KUKA KRL program: EPS_2_25694_GD04_A_20260114065903.src

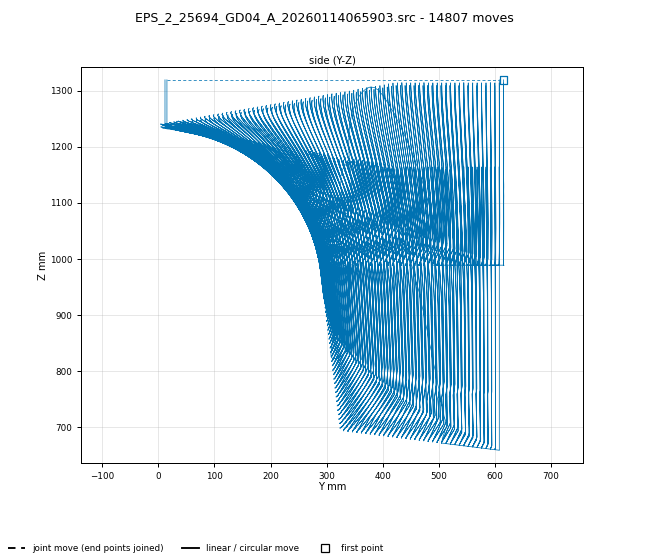
[picture p0: tool path of EPS_2_25694_GD04_A_20260114065903.src, 14807 of 14809 moves have a stored position in this frame; points joined in program order, loops and branches not executed]
&ACCESS RVP
&REL 4
&COMMENT QRS 19112012
&PARAM EDITMASK = *
DEF PART()
EXT BAS (BAS_COMMAND :IN,REAL :IN )
INT I
BAS (#INITMOV,0 )

;KUKA QRS Post kuka4.cps  Date:22-06-2017 !

File_ID=2971

QRS_PRE_INIT()

;Init var - Until changes are made in qrs_pre_init
Outlet_Square_prg=0
Inlet_1_Square_prg=0
Inlet_2_Square_prg=0
Inlet_3_Square_prg=0
Inlet_4_Square_prg=0
Inlet_5_Square_prg=0

Outlet_1={X 0.000, Y 425.000, Z 1043.000, B 0.000, E1 0.000 }
Inlet_1={X 0.000, Y 425.000, Z 703.000, B 0.000, E1 180.000 }
Outlet_1_type=533
Inlet_1_type=533
;QRS#1=Sidecore dimensions
;QRS#2=525-21" Concrete
;QRS#3=525-21" Concrete
;QRS#4=
;QRS#5=
;QRS#6=
;QRS#7=
;QRS#8=
;QRS#9=S306-32
;QRS#10=S306-32
;QRS#11=
;QRS#12=
;QRS#13=
;QRS#14=
;QRS#15=
;QRS#16=1220x127x1676 5,5'
;QRS#17=EPS Height
;QRS#18=1309,5
;QRS#19=*
;QRS#20= UPDATED VERSION 22-06-2017
;QRS#21=*
Outlet_Square=0250
Inlet_1_Square=0250
Inlet_2_Square=0
Inlet_3_Square=0
Inlet_4_Square=0
Inlet_5_Square=0
Mill_Square=1
Outlet_Square_Prg=263
Inlet_1_Square_prg=263

QRS_INIT()

$ADVANCE=5

; T1
PTP {E1 172.608,E2 172.608}
PTP {X 0,Y 615.419,A -85,B 0,C 180,E1 172.608,E2 172.608,E3 0,E4 0,E5 0,E6 0}
QRS_SPEED_INIT()
LIN {X 0,Y 615.419,Z 1319.5,A -85,B 0,C 180,E1 172.608,E2 172.608,E3 0,E4 0,E5 0,E6 0} C_VEL
LIN {X 0,Y 615.419,Z 991.03,A -85,B 0,C 180,E1 172.608,E2 172.608} C_VEL
LIN {X 0,Y 615.445,Z 989.03,A -85,B 0,C 180,E1 172.794,E2 172.794} C_VEL
LIN {X 0,Y 615.855,Z 989.03,A -85,B 0,C 180,E1 174.193,E2 174.193} C_VEL
LIN {X 0,Y 615.875,Z 989.03,A -85,B 0,C 180,E1 178.841,E2 178.841} C_VEL
LIN {X 0,Y 615.861,Z 989.03,A -85,B 0,C 180,E1 183.48,E2 183.48} C_VEL
LIN {X 0,Y 615.852,Z 989.03,A -85,B 0,C 180,E1 188.143,E2 188.143} C_VEL
LIN {X 0,Y 615.813,Z 989.03,A -85,B 0,C 180,E1 192.861,E2 192.861} C_VEL
LIN {X 0,Y 615.807,Z 989.03,A -85,B 0,C 180,E1 197.67,E2 197.67} C_VEL
LIN {X 0,Y 615.805,Z 989.03,A -85,B 0,C 180,E1 198.001,E2 198.001} C_VEL
LIN {X 0,Y 615.77,Z 989.03,A -85,B 0,C 180,E1 202.613,E2 202.613} C_VEL
LIN {X 0,Y 615.246,Z 989.03,A -85,B 0,C 180,E1 205.172,E2 205.172} C_VEL
LIN {X 0,Y 615.74,Z 989.03,A -85,B 0,C 180,E1 207.741,E2 207.741} C_VEL
LIN {X 0,Y 615.245,Z 989.03,A -85,B 0,C 180,E1 210.422,E2 210.422} C_VEL
LIN {X 0,Y 615.834,Z 989.03,A -85,B 0,C 180,E1 213.117,E2 213.117} C_VEL
LIN {X 0,Y 615.539,Z 989.03,A -85,B 0,C 180,E1 215.951,E2 215.951} C_VEL
LIN {X 0,Y 615.602,Z 989.03,A -85,B 0,C 180,E1 217.868,E2 217.868} C_VEL
LIN {X 0,Y 615.676,Z 989.03,A -85,B 0,C 180,E1 221.907,E2 221.907} C_VEL
LIN {X 0,Y 615.231,Z 989.03,A -85,B 0,C 180,E1 225.147,E2 225.147} C_VEL
LIN {X 0,Y 615.682,Z 989.03,A -85,B 0,C 180,E1 228.095,E2 228.095} C_VEL
LIN {X 0,Y 615.612,Z 989.03,A -85,B 0,C 180,E1 232.134,E2 232.134} C_VEL
LIN {X 0,Y 615.586,Z 989.03,A -85,B 0,C 180,E1 234.054,E2 234.054} C_VEL
LIN {X 0,Y 615.729,Z 989.03,A -85,B 0,C 180,E1 236.076,E2 236.076} C_VEL
LIN {X 0,Y 615.766,Z 989.03,A -85,B 0,C 180,E1 236.881,E2 236.881} C_VEL
LIN {X 0,Y 615.665,Z 989.03,A -85,B 0,C 180,E1 239.603,E2 239.603} C_VEL
LIN {X 0,Y 615.571,Z 989.03,A -85,B 0,C 180,E1 240.51,E2 240.51} C_VEL
LIN {X 0,Y 615.286,Z 989.03,A -85,B 0,C 180,E1 240.561,E2 240.561} C_VEL
LIN {X 0,Y 615.222,Z 991.746,A -85,B 0,C 180,E1 240.607,E2 240.607} C_VEL
LIN {X 0,Y 615.448,Z 1058.521,A -85,B 0,C 180,E1 241.501,E2 241.501} C_VEL
LIN {X 0,Y 615.53,Z 1069.288,A -85,B 0,C 180,E1 241.68,E2 241.68} C_VEL
LIN {X 0,Y 615.536,Z 1083.605,A -85,B 0,C 180,E1 241.986,E2 241.986} C_VEL
LIN {X 0,Y 615.507,Z 1092.707,A -85,B 0,C 180,E1 242.216,E2 242.216} C_VEL
LIN {X 0,Y 615.685,Z 1108.532,A -85,B 0,C 180,E1 242.707,E2 242.707} C_VEL
LIN {X 0,Y 615.645,Z 1120.963,A -85,B 0,C 180,E1 243.153,E2 243.153} C_VEL
LIN {X 0,Y 615.565,Z 1130.88,A -85,B 0,C 180,E1 243.554,E2 243.554} C_VEL
LIN {X 0,Y 615.702,Z 1146.604,A -85,B 0,C 180,E1 244.287,E2 244.287} C_VEL
LIN {X 0,Y 615.674,Z 1158.954,A -85,B 0,C 180,E1 244.936,E2 244.936} C_VEL
LIN {X 0,Y 615.686,Z 1170.579,A -85,B 0,C 180,E1 245.615,E2 245.615} C_VEL
LIN {X 0,Y 615.71,Z 1182.431,A -85,B 0,C 180,E1 246.381,E2 246.381} C_VEL
LIN {X 0,Y 615.719,Z 1193.096,A -85,B 0,C 180,E1 247.136,E2 247.136} C_VEL
LIN {X 0,Y 615.717,Z 1204.396,A -85,B 0,C 180,E1 248.013,E2 248.013} C_VEL
LIN {X 0,Y 615.705,Z 1213.657,A -85,B 0,C 180,E1 248.792,E2 248.792} C_VEL
LIN {X 0,Y 615.754,Z 1223.794,A -85,B 0,C 180,E1 249.723,E2 249.723} C_VEL
LIN {X 0,Y 615.723,Z 1233.057,A -85,B 0,C 180,E1 250.647,E2 250.647} C_VEL
LIN {X 0,Y 615.68,Z 1241.424,A -85,B 0,C 180,E1 251.549,E2 251.549} C_VEL
LIN {X 0,Y 615.758,Z 1249.778,A -85,B 0,C 180,E1 252.532,E2 252.532} C_VEL
LIN {X 0,Y 615.711,Z 1257.683,A -85,B 0,C 180,E1 253.542,E2 253.542} C_VEL
LIN {X 0,Y 615.578,Z 1264.428,A -85,B 0,C 180,E1 254.473,E2 254.473} C_VEL
LIN {X 0,Y 615.673,Z 1272.062,A -85,B 0,C 180,E1 255.645,E2 255.645} C_VEL
LIN {X 0,Y 615.813,Z 1277.438,A -85,B 0,C 180,E1 256.544,E2 256.544} C_VEL
LIN {X 0,Y 615.579,Z 1283.91,A -85,B 0,C 180,E1 257.728,E2 257.728} C_VEL
LIN {X 0,Y 615.618,Z 1289.624,A -85,B 0,C 180,E1 258.913,E2 258.913} C_VEL
LIN {X 0,Y 615.829,Z 1294.634,A -85,B 0,C 180,E1 260.096,E2 260.096} C_VEL
LIN {X 0,Y 615.605,Z 1299.063,A -85,B 0,C 180,E1 261.268,E2 261.268} C_VEL
LIN {X 0,Y 615.656,Z 1303.46,A -85,B 0,C 180,E1 262.657,E2 262.657} C_VEL
LIN {X 0,Y 615.79,Z 1306.367,A -85,B 0,C 180,E1 263.748,E2 263.748} C_VEL
LIN {X 0,Y 615.529,Z 1309.384,A -85,B 0,C 180,E1 265.123,E2 265.123} C_VEL
LIN {X 0,Y 615.632,Z 1311.593,A -85,B 0,C 180,E1 266.519,E2 266.519} C_VEL
LIN {X 0,Y 615.819,Z 1312.67,A -85,B 0,C 180,E1 267.449,E2 267.449} C_VEL
LIN {X 0,Y 615.544,Z 1313.716,A -85,B 0,C 180,E1 268.84,E2 268.84} C_VEL
LIN {X 0,Y 615.841,Z 1313.659,A -85,B 0,C 180,E1 271.159,E2 271.159} C_VEL
LIN {X 0,Y 615.625,Z 1313.07,A -85,B 0,C 180,E1 272.088,E2 272.088} C_VEL
LIN {X 0,Y 615.537,Z 1311.611,A -85,B 0,C 180,E1 273.482,E2 273.482} C_VEL
LIN {X 0,Y 615.808,Z 1309.333,A -85,B 0,C 180,E1 274.875,E2 274.875} C_VEL
LIN {X 0,Y 615.603,Z 1306.409,A -85,B 0,C 180,E1 276.25,E2 276.25} C_VEL
LIN {X 0,Y 615.617,Z 1303.276,A -85,B 0,C 180,E1 277.415,E2 277.415} C_VEL
LIN {X 0,Y 615.787,Z 1299.035,A -85,B 0,C 180,E1 278.729,E2 278.729} C_VEL
LIN {X 0,Y 615.576,Z 1294.671,A -85,B 0,C 180,E1 279.908,E2 279.908} C_VEL
LIN {X 0,Y 615.636,Z 1289.622,A -85,B 0,C 180,E1 281.086,E2 281.086} C_VEL
LIN {X 0,Y 615.811,Z 1283.883,A -85,B 0,C 180,E1 282.267,E2 282.267} C_VEL
LIN {X 0,Y 615.629,Z 1277.456,A -85,B 0,C 180,E1 283.46,E2 283.46} C_VEL
LIN {X 0,Y 615.698,Z 1270.195,A -85,B 0,C 180,E1 284.654,E2 284.654} C_VEL
LIN {X 0,Y 615.81,Z 1264.632,A -85,B 0,C 180,E1 285.488,E2 285.488} C_VEL
LIN {X 0,Y 615.663,Z 1255.2,A -85,B 0,C 180,E1 286.791,E2 286.791} C_VEL
LIN {X 0,Y 615.737,Z 1246.606,A -85,B 0,C 180,E1 287.852,E2 287.852} C_VEL
LIN {X 0,Y 615.77,Z 1238.414,A -85,B 0,C 180,E1 288.784,E2 288.784} C_VEL
LIN {X 0,Y 615.695,Z 1228.526,A -85,B 0,C 180,E1 289.816,E2 289.816} C_VEL
LIN {X 0,Y 615.712,Z 1220.54,A -85,B 0,C 180,E1 290.588,E2 290.588} C_VEL
LIN {X 0,Y 615.743,Z 1210.038,A -85,B 0,C 180,E1 291.518,E2 291.518} C_VEL
LIN {X 0,Y 615.702,Z 1200.053,A -85,B 0,C 180,E1 292.335,E2 292.335} C_VEL
LIN {X 0,Y 615.701,Z 1190.291,A -85,B 0,C 180,E1 293.071,E2 293.071} C_VEL
LIN {X 0,Y 615.684,Z 1178.615,A -85,B 0,C 180,E1 293.875,E2 293.875} C_VEL
LIN {X 0,Y 615.706,Z 1166.573,A -85,B 0,C 180,E1 294.624,E2 294.624} C_VEL
LIN {X 0,Y 615.664,Z 1155.895,A -85,B 0,C 180,E1 295.233,E2 295.233} C_VEL
LIN {X 0,Y 615.663,Z 1145.03,A -85,B 0,C 180,E1 295.795,E2 295.795} C_VEL
LIN {X 0,Y 615.698,Z 1130.88,A -85,B 0,C 180,E1 296.439,E2 296.439} C_VEL
LIN {X 0,Y 615.617,Z 1117.679,A -85,B 0,C 180,E1 296.971,E2 296.971} C_VEL
LIN {X 0,Y 615.552,Z 1108.531,A -85,B 0,C 180,E1 297.299,E2 297.299} C_VEL
LIN {X 0,Y 615.614,Z 1091.815,A -85,B 0,C 180,E1 297.801,E2 297.801} C_VEL
LIN {X 0,Y 615.471,Z 1080.012,A -85,B 0,C 180,E1 298.104,E2 298.104} C_VEL
LIN {X 0,Y 615.643,Z 1066.85,A -85,B 0,C 180,E1 298.361,E2 298.361} C_VEL
LIN {X 0,Y 615.612,Z 1048.004,A -85,B 0,C 180,E1 298.638,E2 298.638} C_VEL
LIN {X 0,Y 615.269,Z 989.03,A -85,B 0,C 180,E1 299.434,E2 299.434} C_VEL
LIN {X 0,Y 615.512,Z 989.03,A -85,B 0,C 180,E1 299.476,E2 299.476} C_VEL
LIN {X 0,Y 615.842,Z 989.03,A -85,B 0,C 180,E1 300.388,E2 300.388} C_VEL
LIN {X 0,Y 615.705,Z 989.03,A -85,B 0,C 180,E1 305.938,E2 305.938} C_VEL
LIN {X 0,Y 615.769,Z 989.03,A -85,B 0,C 180,E1 308.853,E2 308.853} C_VEL
LIN {X 0,Y 615.266,Z 989.03,A -85,B 0,C 180,E1 311.939,E2 311.939} C_VEL
LIN {X 0,Y 615.689,Z 989.03,A -85,B 0,C 180,E1 314.896,E2 314.896} C_VEL
LIN {X 0,Y 615.648,Z 989.03,A -85,B 0,C 180,E1 318.494,E2 318.494} C_VEL
LIN {X 0,Y 615.37,Z 989.03,A -85,B 0,C 180,E1 321.115,E2 321.115} C_VEL
LIN {X 0,Y 615.425,Z 989.03,A -85,B 0,C 180,E1 322.154,E2 322.154} C_VEL
LIN {X 0,Y 615.683,Z 989.03,A -85,B 0,C 180,E1 324.059,E2 324.059} C_VEL
LIN {X 0,Y 615.149,Z 989.03,A -85,B 0,C 180,E1 326.842,E2 326.842} C_VEL
LIN {X 0,Y 615.748,Z 989.03,A -85,B 0,C 180,E1 329.606,E2 329.606} C_VEL
LIN {X 0,Y 615.235,Z 989.03,A -85,B 0,C 180,E1 332.234,E2 332.234} C_VEL
LIN {X 0,Y 615.77,Z 989.03,A -85,B 0,C 180,E1 334.851,E2 334.851} C_VEL
LIN {X 0,Y 615.796,Z 989.03,A -85,B 0,C 180,E1 339.878,E2 339.878} C_VEL
LIN {X 0,Y 615.802,Z 989.03,A -85,B 0,C 180,E1 343.784,E2 343.784} C_VEL
LIN {X 0,Y 615.822,Z 989.03,A -85,B 0,C 180,E1 349.507,E2 349.507} C_VEL
LIN {X 0,Y 615.853,Z 989.03,A -85,B 0,C 180,E1 354.193,E2 354.193} C_VEL
LIN {X 0,Y 615.865,Z 989.03,A -85,B 0,C 180,E1 358.841,E2 358.841} C_VEL
LIN {X 0,Y 615.866,Z 989.03,A -85,B 0,C 180,E1 363.48,E2 363.48} C_VEL
LIN {X 0,Y 615.845,Z 989.03,A -85,B 0,C 180,E1 368.143,E2 368.143} C_VEL
LIN {X 0,Y 615.803,Z 989.03,A -85,B 0,C 180,E1 372.862,E2 372.862} C_VEL
LIN {X 0,Y 615.806,Z 989.03,A -85,B 0,C 180,E1 377.67,E2 377.67} C_VEL
LIN {X 0,Y 615.804,Z 989.03,A -85,B 0,C 180,E1 378.001,E2 378.001} C_VEL
LIN {X 0,Y 615.787,Z 989.03,A -85,B 0,C 180,E1 382.612,E2 382.612} C_VEL
LIN {X 0,Y 615.244,Z 989.03,A -85,B 0,C 180,E1 385.172,E2 385.172} C_VEL
LIN {X 0,Y 615.735,Z 989.03,A -85,B 0,C 180,E1 387.741,E2 387.741} C_VEL
LIN {X 0,Y 615.177,Z 989.03,A -85,B 0,C 180,E1 390.425,E2 390.425} C_VEL
LIN {X 0,Y 615.705,Z 989.03,A -85,B 0,C 180,E1 393.124,E2 393.124} C_VEL
LIN {X 0,Y 615.645,Z 989.03,A -85,B 0,C 180,E1 393.916,E2 393.916} C_VEL
LIN {X 0,Y 615.651,Z 989.03,A -85,B 0,C 180,E1 398.864,E2 398.864} C_VEL
LIN {X 0,Y 615.251,Z 989.03,A -85,B 0,C 180,E1 401.943,E2 401.943} C_VEL
LIN {X 0,Y 615.678,Z 989.03,A -85,B 0,C 180,E1 404.897,E2 404.897} C_VEL
LIN {X 0,Y 615.658,Z 989.03,A -85,B 0,C 180,E1 408.496,E2 408.496} C_VEL
LIN {X 0,Y 615.375,Z 989.03,A -85,B 0,C 180,E1 411.117,E2 411.117} C_VEL
LIN {X 0,Y 615.426,Z 989.03,A -85,B 0,C 180,E1 412.156,E2 412.156} C_VEL
LIN {X 0,Y 615.691,Z 989.03,A -85,B 0,C 180,E1 414.061,E2 414.061} C_VEL
LIN {X 0,Y 615.154,Z 989.03,A -85,B 0,C 180,E1 416.844,E2 416.844} C_VEL
LIN {X 0,Y 615.773,Z 989.03,A -85,B 0,C 180,E1 419.609,E2 419.609} C_VEL
LIN {X 0,Y 615.759,Z 989.03,A -85,B 0,C 180,E1 423.303,E2 423.303} C_VEL
LIN {X 0,Y 615.27,Z 989.079,A -85,B 0,C 180,E1 423.866,E2 423.866} C_VEL
LIN {X 0,Y 615.494,Z 997.667,A -85,B 0,C 180,E1 424.288,E2 424.288} C_VEL
LIN {X 0,Y 615.612,Z 1009.734,A -85,B 0,C 180,E1 424.933,E2 424.933} C_VEL
LIN {X 0,Y 615.672,Z 1021.343,A -85,B 0,C 180,E1 425.618,E2 425.618} C_VEL
LIN {X 0,Y 615.7,Z 1032.734,A -85,B 0,C 180,E1 426.357,E2 426.357} C_VEL
LIN {X 0,Y 615.717,Z 1042.488,A -85,B 0,C 180,E1 427.044,E2 427.044} C_VEL
LIN {X 0,Y 615.706,Z 1053.812,A -85,B 0,C 180,E1 427.919,E2 427.919} C_VEL
LIN {X 0,Y 615.708,Z 1064.155,A -85,B 0,C 180,E1 428.792,E2 428.792} C_VEL
LIN {X 0,Y 615.732,Z 1072.675,A -85,B 0,C 180,E1 429.568,E2 429.568} C_VEL
LIN {X 0,Y 615.739,Z 1082.034,A -85,B 0,C 180,E1 430.493,E2 430.493} C_VEL
LIN {X 0,Y 615.681,Z 1089.889,A -85,B 0,C 180,E1 431.327,E2 431.327} C_VEL
LIN {X 0,Y 615.735,Z 1098.523,A -85,B 0,C 180,E1 432.328,E2 432.328} C_VEL
LIN {X 0,Y 615.758,Z 1106.541,A -85,B 0,C 180,E1 433.341,E2 433.341} C_VEL
LIN {X 0,Y 615.587,Z 1114.528,A -85,B 0,C 180,E1 434.443,E2 434.443} C_VEL
LIN {X 0,Y 615.629,Z 1120.5,A -85,B 0,C 180,E1 435.344,E2 435.344} C_VEL
LIN {X 0,Y 615.814,Z 1127.695,A -85,B 0,C 180,E1 436.544,E2 436.544} C_VEL
LIN {X 0,Y 615.591,Z 1134.13,A -85,B 0,C 180,E1 437.729,E2 437.729} C_VEL
LIN {X 0,Y 615.618,Z 1139.819,A -85,B 0,C 180,E1 438.913,E2 438.913} C_VEL
LIN {X 0,Y 615.817,Z 1144.809,A -85,B 0,C 180,E1 440.096,E2 440.096} C_VEL
LIN {X 0,Y 615.604,Z 1149.222,A -85,B 0,C 180,E1 441.268,E2 441.268} C_VEL
LIN {X 0,Y 615.654,Z 1153.586,A -85,B 0,C 180,E1 442.659,E2 442.659} C_VEL
LIN {X 0,Y 615.797,Z 1156.474,A -85,B 0,C 180,E1 443.747,E2 443.747} C_VEL
LIN {X 0,Y 615.543,Z 1159.456,A -85,B 0,C 180,E1 445.123,E2 445.123} C_VEL
LIN {X 0,Y 615.553,Z 1161.021,A -85,B 0,C 180,E1 446.053,E2 446.053} C_VEL
LIN {X 0,Y 615.633,Z 1161.646,A -85,B 0,C 180,E1 446.519,E2 446.519} C_VEL
LIN {X 0,Y 615.703,Z 1163.087,A -85,B 0,C 180,E1 447.912,E2 447.912} C_VEL
LIN {X 0,Y 615.545,Z 1163.726,A -85,B 0,C 180,E1 448.84,E2 448.84} C_VEL
LIN {X 0,Y 615.84,Z 1163.646,A -85,B 0,C 180,E1 451.159,E2 451.159} C_VEL
LIN {X 0,Y 615.601,Z 1162.656,A -85,B 0,C 180,E1 452.552,E2 452.552} C_VEL
LIN {X 0,Y 615.611,Z 1161.544,A -85,B 0,C 180,E1 453.481,E2 453.481} C_VEL
LIN {X 0,Y 615.797,Z 1159.26,A -85,B 0,C 180,E1 454.875,E2 454.875} C_VEL
LIN {X 0,Y 615.534,Z 1156.318,A -85,B 0,C 180,E1 456.245,E2 456.245} C_VEL
LIN {X 0,Y 615.586,Z 1153.213,A -85,B 0,C 180,E1 457.395,E2 457.395} C_VEL
LIN {X 0,Y 615.789,Z 1148.868,A -85,B 0,C 180,E1 458.729,E2 458.729} C_VEL
LIN {X 0,Y 615.587,Z 1144.486,A -85,B 0,C 180,E1 459.908,E2 459.908} C_VEL
LIN {X 0,Y 615.631,Z 1139.418,A -85,B 0,C 180,E1 461.086,E2 461.086} C_VEL
LIN {X 0,Y 615.804,Z 1133.652,A -85,B 0,C 180,E1 462.267,E2 462.267} C_VEL
LIN {X 0,Y 615.622,Z 1127.187,A -85,B 0,C 180,E1 463.46,E2 463.46} C_VEL
LIN {X 0,Y 615.693,Z 1119.896,A -85,B 0,C 180,E1 464.654,E2 464.654} C_VEL
LIN {X 0,Y 615.77,Z 1112.739,A -85,B 0,C 180,E1 465.717,E2 465.717} C_VEL
LIN {X 0,Y 615.611,Z 1104.213,A -85,B 0,C 180,E1 466.871,E2 466.871} C_VEL
LIN {X 0,Y 615.662,Z 1096.204,A -85,B 0,C 180,E1 467.856,E2 467.856} C_VEL
LIN {X 0,Y 615.759,Z 1088.025,A -85,B 0,C 180,E1 468.781,E2 468.781} C_VEL
LIN {X 0,Y 615.689,Z 1079.643,A -85,B 0,C 180,E1 469.662,E2 469.662} C_VEL
LIN {X 0,Y 615.685,Z 1070.04,A -85,B 0,C 180,E1 470.589,E2 470.589} C_VEL
LIN {X 0,Y 615.724,Z 1059.495,A -85,B 0,C 180,E1 471.519,E2 471.519} C_VEL
LIN {X 0,Y 615.715,Z 1049.452,A -85,B 0,C 180,E1 472.335,E2 472.335} C_VEL
LIN {X 0,Y 615.709,Z 1039.629,A -85,B 0,C 180,E1 473.072,E2 473.072} C_VEL
LIN {X 0,Y 615.662,Z 1027.858,A -85,B 0,C 180,E1 473.878,E2 473.878} C_VEL
LIN {X 0,Y 615.718,Z 1017.248,A -85,B 0,C 180,E1 474.54,E2 474.54} C_VEL
LIN {X 0,Y 615.706,Z 1005.438,A -85,B 0,C 180,E1 475.21,E2 475.21} C_VEL
LIN {X 0,Y 615.597,Z 993.583,A -85,B 0,C 180,E1 475.821,E2 475.821} C_VEL
LIN {X 0,Y 615.42,Z 990.651,A -85,B 0,C 180,E1 475.964,E2 475.964} C_VEL
LIN {X 0,Y 615.152,Z 989.03,A -85,B 0,C 180,E1 476.061,E2 476.061} C_VEL
LIN {X 0,Y 615.489,Z 989.03,A -85,B 0,C 180,E1 476.139,E2 476.139} C_VEL
LIN {X 0,Y 615.881,Z 989.03,A -85,B 0,C 180,E1 476.434,E2 476.434} C_VEL
LIN {X 0,Y 615.828,Z 989.03,A -85,B 0,C 180,E1 477.736,E2 477.736} C_VEL
LIN {X 0,Y 615.182,Z 989.03,A -85,B 0,C 180,E1 480.424,E2 480.424} C_VEL
LIN {X 0,Y 615.708,Z 989.03,A -85,B 0,C 180,E1 483.123,E2 483.123} C_VEL
LIN {X 0,Y 615.642,Z 989.03,A -85,B 0,C 180,E1 483.912,E2 483.912} C_VEL
LIN {X 0,Y 615.656,Z 989.03,A -85,B 0,C 180,E1 488.862,E2 488.862} C_VEL
LIN {X 0,Y 615.249,Z 989.03,A -85,B 0,C 180,E1 491.941,E2 491.941} C_VEL
LIN {X 0,Y 615.661,Z 989.03,A -85,B 0,C 180,E1 494.893,E2 494.893} C_VEL
LIN {X 0,Y 615.652,Z 989.03,A -85,B 0,C 180,E1 498.494,E2 498.494} C_VEL
LIN {X 0,Y 615.375,Z 989.03,A -85,B 0,C 180,E1 501.116,E2 501.116} C_VEL
LIN {X 0,Y 615.419,Z 989.03,A -85,B 0,C 180,E1 502.154,E2 502.154} C_VEL
LIN {X 0,Y 615.689,Z 989.03,A -85,B 0,C 180,E1 504.059,E2 504.059} C_VEL
LIN {X 0,Y 615.154,Z 989.03,A -85,B 0,C 180,E1 506.842,E2 506.842} C_VEL
LIN {X 0,Y 615.751,Z 989.03,A -85,B 0,C 180,E1 509.606,E2 509.606} C_VEL
LIN {X 0,Y 615.246,Z 989.03,A -85,B 0,C 180,E1 512.235,E2 512.235} C_VEL
LIN {X 0,Y 615.777,Z 989.03,A -85,B 0,C 180,E1 514.851,E2 514.851} C_VEL
LIN {X 0,Y 615.807,Z 989.03,A -85,B 0,C 180,E1 519.879,E2 519.879} C_VEL
LIN {X 0,Y 615.758,Z 989.03,A -85,B 0,C 180,E1 523.299,E2 523.299} C_VEL
LIN {X 0,Y 615.415,Z 989.03,A -85,B 0,C 180,E1 524.738,E2 524.738} C_VEL
LIN {X 0,Y 615.826,Z 989.03,A -85,B 0,C 180,E1 529.507,E2 529.507} C_VEL
LIN {X 0,Y 615.445,Z 989.03,A -85,B 0,C 180,E1 532.794,E2 532.794} C_VEL
LIN {X 0,Y 613.023,Z 989.03,A -85,B 0,C 180,E1 533.996,E2 533.996} C_VEL
LIN {X 0,Y 607.607,Z 989.03,A -85,B 0,C 180,E1 535.793,E2 535.793} C_VEL
LIN {X 0,Y 607.497,Z 989.03,A -85,B 0,C 180,E1 536.001,E2 536.001} C_VEL
LIN {X 0,Y 607.621,Z 989.03,A -85,B 0,C 180,E1 540,E2 540} C_VEL
LIN {X 0,Y 607.699,Z 989.03,A -85,B 0,C 180,E1 544.272,E2 544.272} C_VEL
LIN {X 0,Y 607.796,Z 989.03,A -85,B 0,C 180,E1 548.567,E2 548.567} C_VEL
LIN {X 0,Y 607.904,Z 989.03,A -85,B 0,C 180,E1 552.909,E2 552.909} C_VEL
LIN {X 0,Y 607.63,Z 989.03,A -85,B 0,C 180,E1 558.834,E2 558.834} C_VEL
LIN {X 0,Y 607.589,Z 989.03,A -85,B 0,C 180,E1 563.413,E2 563.413} C_VEL
LIN {X 0,Y 607.696,Z 989.03,A -85,B 0,C 180,E1 568.15,E2 568.15} C_VEL
LIN {X 0,Y 607.93,Z 989.03,A -85,B 0,C 180,E1 573.097,E2 573.097} C_VEL
LIN {X 0,Y 607.556,Z 989.03,A -85,B 0,C 180,E1 578.382,E2 578.382} C_VEL
LIN {X 0,Y 607.691,Z 989.03,A -85,B 0,C 180,E1 582.1,E2 582.1} C_VEL
LIN {X 0,Y 607.775,Z 989.03,A -85,B 0,C 180,E1 588.144,E2 588.144} C_VEL
LIN {X 0,Y 607.625,Z 989.03,A -85,B 0,C 180,E1 593.413,E2 593.413} C_VEL
LIN {X 0,Y 607.652,Z 989.03,A -85,B 0,C 180,E1 598.566,E2 598.566} C_VEL
LIN {X 0,Y 607.709,Z 989.03,A -85,B 0,C 180,E1 600.165,E2 600.165} C_VEL
LIN {X 0,Y 608.575,Z 1077.126,A -85,B 0,C 180,E1 601.489,E2 601.489} C_VEL
LIN {X 0,Y 608.555,Z 1114.756,A -85,B 0,C 180,E1 602.585,E2 602.585} C_VEL
LIN {X 0,Y 608.428,Z 1150.792,A -85,B 0,C 180,E1 604.177,E2 604.177} C_VEL
LIN {X 0,Y 608.274,Z 1185.935,A -85,B 0,C 180,E1 606.322,E2 606.322} C_VEL
LIN {X 0,Y 608.111,Z 1217.995,A -85,B 0,C 180,E1 608.911,E2 608.911} C_VEL
LIN {X 0,Y 607.969,Z 1246.718,A -85,B 0,C 180,E1 611.925,E2 611.925} C_VEL
LIN {X 0,Y 607.835,Z 1271.188,A -85,B 0,C 180,E1 615.295,E2 615.295} C_VEL
LIN {X 0,Y 607.763,Z 1290.437,A -85,B 0,C 180,E1 618.905,E2 618.905} C_VEL
LIN {X 0,Y 607.783,Z 1303.716,A -85,B 0,C 180,E1 622.51,E2 622.51} C_VEL
LIN {X 0,Y 607.66,Z 1310.955,A -85,B 0,C 180,E1 625.727,E2 625.727} C_VEL
LIN {X 0,Y 607.699,Z 1314.085,A -85,B 0,C 180,E1 628.577,E2 628.577} C_VEL
LIN {X 0,Y 607.887,Z 1314.086,A -85,B 0,C 180,E1 631.422,E2 631.422} C_VEL
LIN {X 0,Y 607.907,Z 1309.758,A -85,B 0,C 180,E1 634.984,E2 634.984} C_VEL
LIN {X 0,Y 607.881,Z 1299.074,A -85,B 0,C 180,E1 638.925,E2 638.925} C_VEL
LIN {X 0,Y 607.91,Z 1283.453,A -85,B 0,C 180,E1 642.544,E2 642.544} C_VEL
LIN {X 0,Y 607.956,Z 1262.352,A -85,B 0,C 180,E1 646.029,E2 646.029} C_VEL
LIN {X 0,Y 608.033,Z 1236.204,A -85,B 0,C 180,E1 649.27,E2 649.27} C_VEL
LIN {X 0,Y 608.169,Z 1206.028,A -85,B 0,C 180,E1 652.137,E2 652.137} C_VEL
LIN {X 0,Y 608.322,Z 1172.896,A -85,B 0,C 180,E1 654.55,E2 654.55} C_VEL
LIN {X 0,Y 608.503,Z 1136.751,A -85,B 0,C 180,E1 656.511,E2 656.511} C_VEL
LIN {X 0,Y 608.582,Z 1099.984,A -85,B 0,C 180,E1 657.91,E2 657.91} C_VEL
LIN {X 0,Y 608.716,Z 1064.141,A -85,B 0,C 180,E1 658.756,E2 658.756} C_VEL
LIN {X 0,Y 607.728,Z 989.475,A -85,B 0,C 180,E1 659.822,E2 659.822} C_VEL
LIN {X 0,Y 607.714,Z 989.03,A -85,B 0,C 180,E1 666.579,E2 666.579} C_VEL
LIN {X 0,Y 607.344,Z 989.03,A -85,B 0,C 180,E1 672.132,E2 672.132} C_VEL
LIN {X 0,Y 607.668,Z 989.03,A -85,B 0,C 180,E1 678.157,E2 678.157} C_VEL
LIN {X 0,Y 607.639,Z 989.03,A -85,B 0,C 180,E1 683.417,E2 683.417} C_VEL
LIN {X 0,Y 607.57,Z 989.03,A -85,B 0,C 180,E1 690.375,E2 690.375} C_VEL
LIN {X 0,Y 607.806,Z 989.03,A -85,B 0,C 180,E1 695.036,E2 695.036} C_VEL
LIN {X 0,Y 607.665,Z 989.03,A -85,B 0,C 180,E1 700.673,E2 700.673} C_VEL
LIN {X 0,Y 607.268,Z 989.03,A -85,B 0,C 180,E1 705.612,E2 705.612} C_VEL
LIN {X 0,Y 607.749,Z 989.03,A -85,B 0,C 180,E1 709.991,E2 709.991} C_VEL
LIN {X 0,Y 607.925,Z 989.03,A -85,B 0,C 180,E1 714.302,E2 714.302} C_VEL
LIN {X 0,Y 607.586,Z 989.03,A -85,B 0,C 180,E1 720,E2 720} C_VEL
LIN {X 0,Y 607.674,Z 989.03,A -85,B 0,C 180,E1 724.272,E2 724.272} C_VEL
LIN {X 0,Y 607.794,Z 989.03,A -85,B 0,C 180,E1 728.567,E2 728.567} C_VEL
LIN {X 0,Y 607.876,Z 989.03,A -85,B 0,C 180,E1 732.909,E2 732.909} C_VEL
LIN {X 0,Y 607.604,Z 989.03,A -85,B 0,C 180,E1 738.835,E2 738.835} C_VEL
LIN {X 0,Y 607.594,Z 989.03,A -85,B 0,C 180,E1 743.413,E2 743.413} C_VEL
LIN {X 0,Y 607.67,Z 989.03,A -85,B 0,C 180,E1 748.151,E2 748.151} C_VEL
LIN {X 0,Y 607.806,Z 989.03,A -85,B 0,C 180,E1 753.105,E2 753.105} C_VEL
LIN {X 0,Y 607.48,Z 989.03,A -85,B 0,C 180,E1 759.642,E2 759.642} C_VEL
LIN {X 0,Y 607.554,Z 989.03,A -85,B 0,C 180,E1 765.938,E2 765.938} C_VEL
LIN {X 0,Y 607.425,Z 989.03,A -85,B 0,C 180,E1 770.362,E2 770.362} C_VEL
LIN {X 0,Y 607.428,Z 989.03,A -85,B 0,C 180,E1 775.154,E2 775.154} C_VEL
LIN {X 0,Y 607.687,Z 989.03,A -85,B 0,C 180,E1 780.352,E2 780.352} C_VEL
LIN {X 0,Y 607.651,Z 989.82,A -85,B 0,C 180,E1 783.548,E2 783.548} C_VEL
LIN {X 0,Y 608.277,Z 1025.109,A -85,B 0,C 180,E1 785.545,E2 785.545} C_VEL
LIN {X 0,Y 608.154,Z 1058.841,A -85,B 0,C 180,E1 788.054,E2 788.054} C_VEL
LIN {X 0,Y 607.98,Z 1089.393,A -85,B 0,C 180,E1 791.027,E2 791.027} C_VEL
LIN {X 0,Y 607.797,Z 1115.33,A -85,B 0,C 180,E1 794.355,E2 794.355} C_VEL
LIN {X 0,Y 607.772,Z 1133.695,A -85,B 0,C 180,E1 797.453,E2 797.453} C_VEL
LIN {X 0,Y 607.781,Z 1149.241,A -85,B 0,C 180,E1 801.073,E2 801.073} C_VEL
LIN {X 0,Y 607.774,Z 1158.319,A -85,B 0,C 180,E1 804.301,E2 804.301} C_VEL
LIN {X 0,Y 607.769,Z 1162.96,A -85,B 0,C 180,E1 807.154,E2 807.154} C_VEL
LIN {X 0,Y 607.73,Z 1164.496,A -85,B 0,C 180,E1 810.001,E2 810.001} C_VEL
LIN {X 0,Y 607.709,Z 1162.852,A -85,B 0,C 180,E1 812.847,E2 812.847} C_VEL
LIN {X 0,Y 607.722,Z 1158.121,A -85,B 0,C 180,E1 815.701,E2 815.701} C_VEL
LIN {X 0,Y 607.813,Z 1147.564,A -85,B 0,C 180,E1 819.287,E2 819.287} C_VEL
LIN {X 0,Y 607.839,Z 1131.246,A -85,B 0,C 180,E1 822.911,E2 822.911} C_VEL
LIN {X 0,Y 607.898,Z 1110.686,A -85,B 0,C 180,E1 826.217,E2 826.217} C_VEL
LIN {X 0,Y 608.04,Z 1085.63,A -85,B 0,C 180,E1 829.286,E2 829.286} C_VEL
LIN {X 0,Y 608.175,Z 1055.481,A -85,B 0,C 180,E1 832.138,E2 832.138} C_VEL
LIN {X 0,Y 608.348,Z 1020.67,A -85,B 0,C 180,E1 834.648,E2 834.648} C_VEL
LIN {X 0,Y 607.948,Z 989.03,A -85,B 0,C 180,E1 836.439,E2 836.439} C_VEL
LIN {X 0,Y 607.81,Z 989.03,A -85,B 0,C 180,E1 843.107,E2 843.107} C_VEL
LIN {X 0,Y 607.506,Z 989.03,A -85,B 0,C 180,E1 849.647,E2 849.647} C_VEL
LIN {X 0,Y 607.518,Z 989.03,A -85,B 0,C 180,E1 855.936,E2 855.936} C_VEL
LIN {X 0,Y 607.424,Z 989.03,A -85,B 0,C 180,E1 860.366,E2 860.366} C_VEL
LIN {X 0,Y 607.422,Z 989.03,A -85,B 0,C 180,E1 865.155,E2 865.155} C_VEL
LIN {X 0,Y 607.567,Z 989.03,A -85,B 0,C 180,E1 870.378,E2 870.378} C_VEL
LIN {X 0,Y 607.799,Z 989.03,A -85,B 0,C 180,E1 875.036,E2 875.036} C_VEL
LIN {X 0,Y 607.663,Z 989.03,A -85,B 0,C 180,E1 881.167,E2 881.167} C_VEL
LIN {X 0,Y 607.249,Z 989.03,A -85,B 0,C 180,E1 885.733,E2 885.733} C_VEL
LIN {X 0,Y 607.754,Z 989.03,A -85,B 0,C 180,E1 889.991,E2 889.991} C_VEL
LIN {X 0,Y 607.909,Z 989.03,A -85,B 0,C 180,E1 894.302,E2 894.302} C_VEL
LIN {X 0,Y 607.497,Z 989.03,A -85,B 0,C 180,E1 896.001,E2 896.001} C_VEL
LIN {X 0,Y 603.696,Z 989.03,A -85,B 0,C 180,E1 897.613,E2 897.613} C_VEL
LIN {X 0,Y 599.806,Z 989.03,A -85,B 0,C 180,E1 899.244,E2 899.244} C_VEL
LIN {X 0,Y 599.78,Z 989.03,A -85,B 0,C 180,E1 904.329,E2 904.329} C_VEL
LIN {X 0,Y 599.852,Z 989.03,A -85,B 0,C 180,E1 908.681,E2 908.681} C_VEL
LIN {X 0,Y 599.925,Z 989.03,A -85,B 0,C 180,E1 913.083,E2 913.083} C_VEL
LIN {X 0,Y 599.672,Z 989.03,A -85,B 0,C 180,E1 919.094,E2 919.094} C_VEL
LIN {X 0,Y 599.598,Z 989.03,A -85,B 0,C 180,E1 923.744,E2 923.744} C_VEL
LIN {X 0,Y 599.687,Z 989.03,A -85,B 0,C 180,E1 928.56,E2 928.56} C_VEL
LIN {X 0,Y 599.814,Z 989.03,A -85,B 0,C 180,E1 933.878,E2 933.878} C_VEL
LIN {X 0,Y 599.539,Z 989.03,A -85,B 0,C 180,E1 938.992,E2 938.992} C_VEL
LIN {X 0,Y 599.496,Z 989.03,A -85,B 0,C 180,E1 943.115,E2 943.115} C_VEL
LIN {X 0,Y 599.595,Z 989.03,A -85,B 0,C 180,E1 949.129,E2 949.129} C_VEL
LIN {X 0,Y 599.717,Z 989.03,A -85,B 0,C 180,E1 954.638,E2 954.638} C_VEL
LIN {X 0,Y 599.889,Z 989.522,A -85,B 0,C 180,E1 959.748,E2 959.748} C_VEL
LIN {X 0,Y 601.492,Z 997.227,A -85,B 0,C 180,E1 959.942,E2 959.942} C_VEL
LIN {X 0,Y 601.63,Z 1077.166,A -85,B 0,C 180,E1 961.13,E2 961.13} C_VEL
LIN {X 0,Y 601.497,Z 1113.617,A -85,B 0,C 180,E1 962.194,E2 962.194} C_VEL
LIN {X 0,Y 601.209,Z 1148.932,A -85,B 0,C 180,E1 963.744,E2 963.744} C_VEL
LIN {X 0,Y 600.865,Z 1184.565,A -85,B 0,C 180,E1 965.914,E2 965.914} C_VEL
LIN {X 0,Y 600.542,Z 1217.043,A -85,B 0,C 180,E1 968.544,E2 968.544} C_VEL
LIN {X 0,Y 600.234,Z 1245.115,A -85,B 0,C 180,E1 971.494,E2 971.494} C_VEL
LIN {X 0,Y 599.993,Z 1269.748,A -85,B 0,C 180,E1 974.874,E2 974.874} C_VEL
LIN {X 0,Y 599.872,Z 1288.763,A -85,B 0,C 180,E1 978.39,E2 978.39} C_VEL
LIN {X 0,Y 599.857,Z 1301.445,A -85,B 0,C 180,E1 981.683,E2 981.683} C_VEL
LIN {X 0,Y 599.777,Z 1309.755,A -85,B 0,C 180,E1 984.948,E2 984.948} C_VEL
LIN {X 0,Y 599.8,Z 1314.085,A -85,B 0,C 180,E1 988.558,E2 988.558} C_VEL
LIN {X 0,Y 599.98,Z 1314.086,A -85,B 0,C 180,E1 991.441,E2 991.441} C_VEL
LIN {X 0,Y 599.994,Z 1309.758,A -85,B 0,C 180,E1 995.05,E2 995.05} C_VEL
LIN {X 0,Y 599.98,Z 1299.074,A -85,B 0,C 180,E1 999.044,E2 999.044} C_VEL
LIN {X 0,Y 600.044,Z 1283.454,A -85,B 0,C 180,E1 1002.711,E2 1002.711} C_VEL
LIN {X 0,Y 600.116,Z 1261.717,A -85,B 0,C 180,E1 1006.334,E2 1006.334} C_VEL
LIN {X 0,Y 600.366,Z 1236.03,A -85,B 0,C 180,E1 1009.545,E2 1009.545} C_VEL
LIN {X 0,Y 600.635,Z 1205.455,A -85,B 0,C 180,E1 1012.479,E2 1012.479} C_VEL
LIN {X 0,Y 601.015,Z 1170.879,A -85,B 0,C 180,E1 1015.001,E2 1015.001} C_VEL
LIN {X 0,Y 601.365,Z 1132.84,A -85,B 0,C 180,E1 1017.036,E2 1017.036} C_VEL
LIN {X 0,Y 601.577,Z 1093.56,A -85,B 0,C 180,E1 1018.463,E2 1018.463} C_VEL
LIN {X 0,Y 601.808,Z 1054.486,A -85,B 0,C 180,E1 1019.271,E2 1019.271} C_VEL
LIN {X 0,Y 600.801,Z 992.559,A -85,B 0,C 180,E1 1020.16,E2 1020.16} C_VEL
LIN {X 0,Y 599.984,Z 989.03,A -85,B 0,C 180,E1 1020.319,E2 1020.319} C_VEL
LIN {X 0,Y 599.762,Z 989.03,A -85,B 0,C 180,E1 1027.145,E2 1027.145} C_VEL
LIN {X 0,Y 599.439,Z 989.03,A -85,B 0,C 180,E1 1033.113,E2 1033.113} C_VEL
LIN {X 0,Y 599.592,Z 989.03,A -85,B 0,C 180,E1 1039.026,E2 1039.026} C_VEL
LIN {X 0,Y 599.566,Z 989.03,A -85,B 0,C 180,E1 1044.63,E2 1044.63} C_VEL
LIN {X 0,Y 599.633,Z 989.03,A -85,B 0,C 180,E1 1049.782,E2 1049.782} C_VEL
LIN {X 0,Y 599.868,Z 989.03,A -85,B 0,C 180,E1 1054.904,E2 1054.904} C_VEL
LIN {X 0,Y 599.739,Z 989.03,A -85,B 0,C 180,E1 1060.908,E2 1060.908} C_VEL
LIN {X 0,Y 599.404,Z 989.03,A -85,B 0,C 180,E1 1065.419,E2 1065.419} C_VEL
LIN {X 0,Y 599.808,Z 989.03,A -85,B 0,C 180,E1 1069.857,E2 1069.857} C_VEL
LIN {X 0,Y 600.023,Z 989.03,A -85,B 0,C 180,E1 1074.227,E2 1074.227} C_VEL
LIN {X 0,Y 599.685,Z 989.03,A -85,B 0,C 180,E1 1080,E2 1080} C_VEL
LIN {X 0,Y 599.757,Z 989.03,A -85,B 0,C 180,E1 1084.329,E2 1084.329} C_VEL
LIN {X 0,Y 599.85,Z 989.03,A -85,B 0,C 180,E1 1088.681,E2 1088.681} C_VEL
LIN {X 0,Y 599.903,Z 989.03,A -85,B 0,C 180,E1 1093.084,E2 1093.084} C_VEL
LIN {X 0,Y 599.665,Z 989.03,A -85,B 0,C 180,E1 1099.094,E2 1099.094} C_VEL
LIN {X 0,Y 599.606,Z 989.03,A -85,B 0,C 180,E1 1103.744,E2 1103.744} C_VEL
LIN {X 0,Y 599.662,Z 989.03,A -85,B 0,C 180,E1 1108.561,E2 1108.561} C_VEL
LIN {X 0,Y 599.678,Z 989.03,A -85,B 0,C 180,E1 1113.861,E2 1113.861} C_VEL
LIN {X 0,Y 599.594,Z 989.03,A -85,B 0,C 180,E1 1118.988,E2 1118.988} C_VEL
LIN {X 0,Y 599.557,Z 989.03,A -85,B 0,C 180,E1 1125.193,E2 1125.193} C_VEL
LIN {X 0,Y 599.531,Z 989.03,A -85,B 0,C 180,E1 1131.006,E2 1131.006} C_VEL
LIN {X 0,Y 599.563,Z 989.03,A -85,B 0,C 180,E1 1134.629,E2 1134.629} C_VEL
LIN {X 0,Y 599.708,Z 989.03,A -85,B 0,C 180,E1 1139.785,E2 1139.785} C_VEL
LIN {X 0,Y 599.913,Z 989.812,A -85,B 0,C 180,E1 1143.18,E2 1143.18} C_VEL
LIN {X 0,Y 600.997,Z 1016.313,A -85,B 0,C 180,E1 1144.671,E2 1144.671} C_VEL
LIN {X 0,Y 600.696,Z 1051.951,A -85,B 0,C 180,E1 1147.18,E2 1147.18} C_VEL
LIN {X 0,Y 600.392,Z 1083.053,A -85,B 0,C 180,E1 1150.087,E2 1150.087} C_VEL
LIN {X 0,Y 600.189,Z 1109.946,A -85,B 0,C 180,E1 1153.374,E2 1153.374} C_VEL
LIN {X 0,Y 600.099,Z 1129.787,A -85,B 0,C 180,E1 1156.553,E2 1156.553} C_VEL
LIN {X 0,Y 600.012,Z 1146.562,A -85,B 0,C 180,E1 1160.227,E2 1160.227} C_VEL
LIN {X 0,Y 599.964,Z 1157.365,A -85,B 0,C 180,E1 1163.781,E2 1163.781} C_VEL
LIN {X 0,Y 599.875,Z 1162.959,A -85,B 0,C 180,E1 1167.117,E2 1167.117} C_VEL
LIN {X 0,Y 599.83,Z 1164.496,A -85,B 0,C 180,E1 1170.001,E2 1170.001} C_VEL
LIN {X 0,Y 599.824,Z 1162.853,A -85,B 0,C 180,E1 1172.885,E2 1172.885} C_VEL
LIN {X 0,Y 599.763,Z 1157.099,A -85,B 0,C 180,E1 1176.254,E2 1176.254} C_VEL
LIN {X 0,Y 599.852,Z 1146.228,A -85,B 0,C 180,E1 1179.777,E2 1179.777} C_VEL
LIN {X 0,Y 599.974,Z 1129.305,A -85,B 0,C 180,E1 1183.451,E2 1183.451} C_VEL
LIN {X 0,Y 600.104,Z 1106.532,A -85,B 0,C 180,E1 1187.02,E2 1187.02} C_VEL
LIN {X 0,Y 600.376,Z 1078.917,A -85,B 0,C 180,E1 1190.259,E2 1190.259} C_VEL
LIN {X 0,Y 600.72,Z 1047.546,A -85,B 0,C 180,E1 1193.075,E2 1193.075} C_VEL
LIN {X 0,Y 601.07,Z 1014.487,A -85,B 0,C 180,E1 1195.344,E2 1195.344} C_VEL
LIN {X 0,Y 600.12,Z 990.014,A -85,B 0,C 180,E1 1196.71,E2 1196.71} C_VEL
LIN {X 0,Y 600.006,Z 989.03,A -85,B 0,C 180,E1 1196.918,E2 1196.918} C_VEL
LIN {X 0,Y 599.678,Z 989.03,A -85,B 0,C 180,E1 1203.864,E2 1203.864} C_VEL
LIN {X 0,Y 599.607,Z 989.03,A -85,B 0,C 180,E1 1208.989,E2 1208.989} C_VEL
LIN {X 0,Y 599.534,Z 989.03,A -85,B 0,C 180,E1 1215.193,E2 1215.193} C_VEL
LIN {X 0,Y 599.53,Z 989.03,A -85,B 0,C 180,E1 1221.007,E2 1221.007} C_VEL
LIN {X 0,Y 599.557,Z 989.03,A -85,B 0,C 180,E1 1224.63,E2 1224.63} C_VEL
LIN {X 0,Y 599.634,Z 989.03,A -85,B 0,C 180,E1 1229.782,E2 1229.782} C_VEL
LIN {X 0,Y 599.874,Z 989.03,A -85,B 0,C 180,E1 1234.905,E2 1234.905} C_VEL
LIN {X 0,Y 599.792,Z 989.03,A -85,B 0,C 180,E1 1240.91,E2 1240.91} C_VEL
LIN {X 0,Y 599.409,Z 989.03,A -85,B 0,C 180,E1 1245.42,E2 1245.42} C_VEL
LIN {X 0,Y 599.812,Z 989.03,A -85,B 0,C 180,E1 1249.857,E2 1249.857} C_VEL
LIN {X 0,Y 600.012,Z 989.03,A -85,B 0,C 180,E1 1254.227,E2 1254.227} C_VEL
LIN {X 0,Y 599.806,Z 989.03,A -85,B 0,C 180,E1 1259.244,E2 1259.244} C_VEL
LIN {X 0,Y 595.646,Z 989.03,A -85,B 0,C 180,E1 1260.875,E2 1260.875} C_VEL
LIN {X 0,Y 591.828,Z 989.03,A -85,B 0,C 180,E1 1262.527,E2 1262.527} C_VEL
LIN {X 0,Y 591.911,Z 989.03,A -85,B 0,C 180,E1 1268.798,E2 1268.798} C_VEL
LIN {X 0,Y 591.687,Z 989.03,A -85,B 0,C 180,E1 1274.27,E2 1274.27} C_VEL
LIN {X 0,Y 591.712,Z 989.03,A -85,B 0,C 180,E1 1279.361,E2 1279.361} C_VEL
LIN {X 0,Y 591.63,Z 989.03,A -85,B 0,C 180,E1 1284.084,E2 1284.084} C_VEL
LIN {X 0,Y 591.672,Z 989.03,A -85,B 0,C 180,E1 1288.984,E2 1288.984} C_VEL
LIN {X 0,Y 591.884,Z 989.03,A -85,B 0,C 180,E1 1294.116,E2 1294.116} C_VEL
LIN {X 0,Y 591.596,Z 989.03,A -85,B 0,C 180,E1 1300.072,E2 1300.072} C_VEL
LIN {X 0,Y 591.433,Z 989.03,A -85,B 0,C 180,E1 1305.592,E2 1305.592} C_VEL
LIN {X 0,Y 591.591,Z 989.03,A -85,B 0,C 180,E1 1310.379,E2 1310.379} C_VEL
LIN {X 0,Y 591.902,Z 989.03,A -85,B 0,C 180,E1 1315.883,E2 1315.883} C_VEL
LIN {X 0,Y 591.953,Z 989.474,A -85,B 0,C 180,E1 1319.299,E2 1319.299} C_VEL
LIN {X 0,Y 594.68,Z 998.902,A -85,B 0,C 180,E1 1319.584,E2 1319.584} C_VEL
LIN {X 0,Y 594.688,Z 1077.22,A -85,B 0,C 180,E1 1320.762,E2 1320.762} C_VEL
LIN {X 0,Y 594.439,Z 1114.246,A -85,B 0,C 180,E1 1321.858,E2 1321.858} C_VEL
LIN {X 0,Y 594.009,Z 1148.924,A -85,B 0,C 180,E1 1323.4,E2 1323.4} C_VEL
LIN {X 0,Y 593.46,Z 1183.781,A -85,B 0,C 180,E1 1325.536,E2 1325.536} C_VEL
LIN {X 0,Y 592.981,Z 1215.316,A -85,B 0,C 180,E1 1328.093,E2 1328.093} C_VEL
LIN {X 0,Y 592.558,Z 1243.512,A -85,B 0,C 180,E1 1331.053,E2 1331.053} C_VEL
LIN {X 0,Y 592.162,Z 1267.33,A -85,B 0,C 180,E1 1334.29,E2 1334.29} C_VEL
LIN {X 0,Y 592.059,Z 1285.275,A -85,B 0,C 180,E1 1337.487,E2 1337.487} C_VEL
LIN {X 0,Y 592.051,Z 1299.071,A -85,B 0,C 180,E1 1340.833,E2 1340.833} C_VEL
LIN {X 0,Y 592.022,Z 1308.219,A -85,B 0,C 180,E1 1344.148,E2 1344.148} C_VEL
LIN {X 0,Y 592.063,Z 1312.905,A -85,B 0,C 180,E1 1347.078,E2 1347.078} C_VEL
LIN {X 0,Y 591.931,Z 1314.5,A -85,B 0,C 180,E1 1349.999,E2 1349.999} C_VEL
LIN {X 0,Y 591.894,Z 1312.907,A -85,B 0,C 180,E1 1352.922,E2 1352.922} C_VEL
LIN {X 0,Y 591.947,Z 1306.579,A -85,B 0,C 180,E1 1356.593,E2 1356.593} C_VEL
LIN {X 0,Y 591.952,Z 1295.047,A -85,B 0,C 180,E1 1360.279,E2 1360.279} C_VEL
LIN {X 0,Y 592.144,Z 1278.319,A -85,B 0,C 180,E1 1363.867,E2 1363.867} C_VEL
LIN {X 0,Y 592.377,Z 1256.728,A -85,B 0,C 180,E1 1367.267,E2 1367.267} C_VEL
LIN {X 0,Y 592.782,Z 1229.448,A -85,B 0,C 180,E1 1370.522,E2 1370.522} C_VEL
LIN {X 0,Y 593.257,Z 1197.684,A -85,B 0,C 180,E1 1373.417,E2 1373.417} C_VEL
LIN {X 0,Y 593.752,Z 1163.246,A -85,B 0,C 180,E1 1375.799,E2 1375.799} C_VEL
LIN {X 0,Y 594.264,Z 1126.526,A -85,B 0,C 180,E1 1377.658,E2 1377.658} C_VEL
LIN {X 0,Y 594.592,Z 1088.332,A -85,B 0,C 180,E1 1378.967,E2 1378.967} C_VEL
LIN {X 0,Y 594.884,Z 1047.179,A -85,B 0,C 180,E1 1379.745,E2 1379.745} C_VEL
LIN {X 0,Y 594.038,Z 994.993,A -85,B 0,C 180,E1 1380.506,E2 1380.506} C_VEL
LIN {X 0,Y 591.964,Z 989.03,A -85,B 0,C 180,E1 1380.768,E2 1380.768} C_VEL
LIN {X 0,Y 591.834,Z 989.03,A -85,B 0,C 180,E1 1387.779,E2 1387.779} C_VEL
LIN {X 0,Y 591.583,Z 989.03,A -85,B 0,C 180,E1 1394.423,E2 1394.423} C_VEL
LIN {X 0,Y 591.595,Z 989.03,A -85,B 0,C 180,E1 1399.926,E2 1399.926} C_VEL
LIN {X 0,Y 591.65,Z 989.03,A -85,B 0,C 180,E1 1404.702,E2 1404.702} C_VEL
LIN {X 0,Y 591.582,Z 989.03,A -85,B 0,C 180,E1 1411.012,E2 1411.012} C_VEL
LIN {X 0,Y 591.675,Z 989.03,A -85,B 0,C 180,E1 1415.918,E2 1415.918} C_VEL
LIN {X 0,Y 591.837,Z 989.03,A -85,B 0,C 180,E1 1420.643,E2 1420.643} C_VEL
LIN {X 0,Y 591.534,Z 989.03,A -85,B 0,C 180,E1 1425.221,E2 1425.221} C_VEL
LIN {X 0,Y 591.878,Z 989.03,A -85,B 0,C 180,E1 1429.72,E2 1429.72} C_VEL
LIN {X 0,Y 592.086,Z 989.03,A -85,B 0,C 180,E1 1434.149,E2 1434.149} C_VEL
LIN {X 0,Y 591.785,Z 989.03,A -85,B 0,C 180,E1 1440,E2 1440} C_VEL
LIN {X 0,Y 591.842,Z 989.03,A -85,B 0,C 180,E1 1444.387,E2 1444.387} C_VEL
LIN {X 0,Y 591.909,Z 989.03,A -85,B 0,C 180,E1 1448.798,E2 1448.798} C_VEL
LIN {X 0,Y 591.673,Z 989.03,A -85,B 0,C 180,E1 1454.269,E2 1454.269} C_VEL
LIN {X 0,Y 591.723,Z 989.03,A -85,B 0,C 180,E1 1459.361,E2 1459.361} C_VEL
LIN {X 0,Y 591.644,Z 989.03,A -85,B 0,C 180,E1 1464.084,E2 1464.084} C_VEL
LIN {X 0,Y 591.64,Z 989.03,A -85,B 0,C 180,E1 1468.985,E2 1468.985} C_VEL
LIN {X 0,Y 591.726,Z 989.03,A -85,B 0,C 180,E1 1474.126,E2 1474.126} C_VEL
LIN {X 0,Y 591.522,Z 989.03,A -85,B 0,C 180,E1 1480.065,E2 1480.065} C_VEL
LIN {X 0,Y 591.615,Z 989.03,A -85,B 0,C 180,E1 1485.574,E2 1485.574} C_VEL
LIN {X 0,Y 591.577,Z 989.03,A -85,B 0,C 180,E1 1490.38,E2 1490.38} C_VEL
LIN {X 0,Y 591.497,Z 989.03,A -85,B 0,C 180,E1 1495.858,E2 1495.858} C_VEL
LIN {X 0,Y 591.75,Z 989.03,A -85,B 0,C 180,E1 1501.02,E2 1501.02} C_VEL
LIN {X 0,Y 591.901,Z 989.137,A -85,B 0,C 180,E1 1502.755,E2 1502.755} C_VEL
LIN {X 0,Y 593.708,Z 1001.834,A -85,B 0,C 180,E1 1503.499,E2 1503.499} C_VEL
LIN {X 0,Y 593.413,Z 1036.96,A -85,B 0,C 180,E1 1505.721,E2 1505.721} C_VEL
LIN {X 0,Y 592.94,Z 1069.858,A -85,B 0,C 180,E1 1508.474,E2 1508.474} C_VEL
LIN {X 0,Y 592.53,Z 1098.654,A -85,B 0,C 180,E1 1511.63,E2 1511.63} C_VEL
LIN {X 0,Y 592.186,Z 1122.336,A -85,B 0,C 180,E1 1515.049,E2 1515.049} C_VEL
LIN {X 0,Y 591.998,Z 1140.258,A -85,B 0,C 180,E1 1518.517,E2 1518.517} C_VEL
LIN {X 0,Y 591.97,Z 1153.837,A -85,B 0,C 180,E1 1522.31,E2 1522.31} C_VEL
LIN {X 0,Y 591.885,Z 1161.031,A -85,B 0,C 180,E1 1525.614,E2 1525.614} C_VEL
LIN {X 0,Y 591.907,Z 1164.118,A -85,B 0,C 180,E1 1528.54,E2 1528.54} C_VEL
LIN {X 0,Y 592.084,Z 1164.055,A -85,B 0,C 180,E1 1531.461,E2 1531.461} C_VEL
LIN {X 0,Y 592.067,Z 1159.672,A -85,B 0,C 180,E1 1535.118,E2 1535.118} C_VEL
LIN {X 0,Y 592.1,Z 1148.908,A -85,B 0,C 180,E1 1539.166,E2 1539.166} C_VEL
LIN {X 0,Y 592.173,Z 1133.214,A -85,B 0,C 180,E1 1542.884,E2 1542.884} C_VEL
LIN {X 0,Y 592.325,Z 1111.659,A -85,B 0,C 180,E1 1546.518,E2 1546.518} C_VEL
LIN {X 0,Y 592.663,Z 1085.544,A -85,B 0,C 180,E1 1549.818,E2 1549.818} C_VEL
LIN {X 0,Y 593.122,Z 1055.227,A -85,B 0,C 180,E1 1552.755,E2 1552.755} C_VEL
LIN {X 0,Y 593.689,Z 1020.807,A -85,B 0,C 180,E1 1555.291,E2 1555.291} C_VEL
LIN {X 0,Y 593.21,Z 993.376,A -85,B 0,C 180,E1 1556.884,E2 1556.884} C_VEL
LIN {X 0,Y 592.037,Z 989.03,A -85,B 0,C 180,E1 1557.189,E2 1557.189} C_VEL
LIN {X 0,Y 591.727,Z 989.03,A -85,B 0,C 180,E1 1564.128,E2 1564.128} C_VEL
LIN {X 0,Y 591.521,Z 989.03,A -85,B 0,C 180,E1 1570.068,E2 1570.068} C_VEL
LIN {X 0,Y 591.596,Z 989.03,A -85,B 0,C 180,E1 1575.579,E2 1575.579} C_VEL
LIN {X 0,Y 591.579,Z 989.03,A -85,B 0,C 180,E1 1580.381,E2 1580.381} C_VEL
LIN {X 0,Y 591.494,Z 989.03,A -85,B 0,C 180,E1 1585.859,E2 1585.859} C_VEL
LIN {X 0,Y 591.581,Z 989.03,A -85,B 0,C 180,E1 1591.012,E2 1591.012} C_VEL
LIN {X 0,Y 591.676,Z 989.03,A -85,B 0,C 180,E1 1595.918,E2 1595.918} C_VEL
LIN {X 0,Y 591.87,Z 989.03,A -85,B 0,C 180,E1 1600.645,E2 1600.645} C_VEL
LIN {X 0,Y 591.462,Z 989.03,A -85,B 0,C 180,E1 1605.816,E2 1605.816} C_VEL
LIN {X 0,Y 591.679,Z 989.03,A -85,B 0,C 180,E1 1611.198,E2 1611.198} C_VEL
LIN {X 0,Y 591.745,Z 989.03,A -85,B 0,C 180,E1 1615.613,E2 1615.613} C_VEL
LIN {X 0,Y 591.819,Z 989.03,A -85,B 0,C 180,E1 1620,E2 1620} C_VEL
LIN {X 0,Y 591.828,Z 989.03,A -85,B 0,C 180,E1 1622.527,E2 1622.527} C_VEL
LIN {X 0,Y 589.392,Z 989.03,A -85,B 0,C 180,E1 1623.777,E2 1623.777} C_VEL
LIN {X 0,Y 583.903,Z 989.03,A -85,B 0,C 180,E1 1625.646,E2 1625.646} C_VEL
LIN {X 0,Y 583.811,Z 989.03,A -85,B 0,C 180,E1 1625.862,E2 1625.862} C_VEL
LIN {X 0,Y 583.76,Z 989.03,A -85,B 0,C 180,E1 1630.795,E2 1630.795} C_VEL
LIN {X 0,Y 583.709,Z 989.03,A -85,B 0,C 180,E1 1634.982,E2 1634.982} C_VEL
LIN {X 0,Y 583.771,Z 989.03,A -85,B 0,C 180,E1 1639.635,E2 1639.635} C_VEL
LIN {X 0,Y 583.671,Z 989.03,A -85,B 0,C 180,E1 1644.434,E2 1644.434} C_VEL
LIN {X 0,Y 583.689,Z 989.03,A -85,B 0,C 180,E1 1649.419,E2 1649.419} C_VEL
LIN {X 0,Y 583.897,Z 989.03,A -85,B 0,C 180,E1 1654.648,E2 1654.648} C_VEL
LIN {X 0,Y 583.68,Z 989.03,A -85,B 0,C 180,E1 1660.264,E2 1660.264} C_VEL
LIN {X 0,Y 583.637,Z 989.03,A -85,B 0,C 180,E1 1666.379,E2 1666.379} C_VEL
LIN {X 0,Y 583.747,Z 989.03,A -85,B 0,C 180,E1 1671.653,E2 1671.653} C_VEL
LIN {X 0,Y 583.974,Z 989.03,A -85,B 0,C 180,E1 1677.135,E2 1677.135} C_VEL
LIN {X 0,Y 583.997,Z 989.036,A -85,B 0,C 180,E1 1678.828,E2 1678.828} C_VEL
LIN {X 0,Y 587.878,Z 1000.279,A -85,B 0,C 180,E1 1679.213,E2 1679.213} C_VEL
LIN {X 0,Y 587.772,Z 1078.814,A -85,B 0,C 180,E1 1680.418,E2 1680.418} C_VEL
LIN {X 0,Y 587.384,Z 1116.422,A -85,B 0,C 180,E1 1681.571,E2 1681.571} C_VEL
LIN {X 0,Y 586.733,Z 1152.74,A -85,B 0,C 180,E1 1683.254,E2 1683.254} C_VEL
LIN {X 0,Y 586.012,Z 1187.624,A -85,B 0,C 180,E1 1685.489,E2 1685.489} C_VEL
LIN {X 0,Y 585.353,Z 1220.447,A -85,B 0,C 180,E1 1688.283,E2 1688.283} C_VEL
LIN {X 0,Y 584.791,Z 1249.769,A -85,B 0,C 180,E1 1691.572,E2 1691.572} C_VEL
LIN {X 0,Y 584.378,Z 1273.163,A -85,B 0,C 180,E1 1695.035,E2 1695.035} C_VEL
LIN {X 0,Y 584.152,Z 1291.03,A -85,B 0,C 180,E1 1698.596,E2 1698.596} C_VEL
LIN {X 0,Y 584.098,Z 1303.716,A -85,B 0,C 180,E1 1702.204,E2 1702.204} C_VEL
LIN {X 0,Y 583.972,Z 1310.955,A -85,B 0,C 180,E1 1705.553,E2 1705.553} C_VEL
LIN {X 0,Y 584.027,Z 1314.086,A -85,B 0,C 180,E1 1708.519,E2 1708.519} C_VEL
LIN {X 0,Y 584.183,Z 1314.087,A -85,B 0,C 180,E1 1711.48,E2 1711.48} C_VEL
LIN {X 0,Y 584.21,Z 1309.757,A -85,B 0,C 180,E1 1715.186,E2 1715.186} C_VEL
LIN {X 0,Y 584.19,Z 1299.074,A -85,B 0,C 180,E1 1719.29,E2 1719.29} C_VEL
LIN {X 0,Y 584.317,Z 1283.452,A -85,B 0,C 180,E1 1723.059,E2 1723.059} C_VEL
LIN {X 0,Y 584.557,Z 1262.379,A -85,B 0,C 180,E1 1726.686,E2 1726.686} C_VEL
LIN {X 0,Y 585.027,Z 1236.752,A -85,B 0,C 180,E1 1729.998,E2 1729.998} C_VEL
LIN {X 0,Y 585.59,Z 1206.269,A -85,B 0,C 180,E1 1733.018,E2 1733.018} C_VEL
LIN {X 0,Y 586.334,Z 1172.551,A -85,B 0,C 180,E1 1735.56,E2 1735.56} C_VEL
LIN {X 0,Y 587.022,Z 1136.761,A -85,B 0,C 180,E1 1737.562,E2 1737.562} C_VEL
LIN {X 0,Y 587.571,Z 1099.38,A -85,B 0,C 180,E1 1739.021,E2 1739.021} C_VEL
LIN {X 0,Y 588.018,Z 1064.285,A -85,B 0,C 180,E1 1739.866,E2 1739.866} C_VEL
LIN {X 0,Y 587.204,Z 997.338,A -85,B 0,C 180,E1 1740.867,E2 1740.867} C_VEL
LIN {X 0,Y 583.868,Z 989.03,A -85,B 0,C 180,E1 1741.232,E2 1741.232} C_VEL
LIN {X 0,Y 583.834,Z 989.03,A -85,B 0,C 180,E1 1746.754,E2 1746.754} C_VEL
LIN {X 0,Y 583.585,Z 989.03,A -85,B 0,C 180,E1 1752.244,E2 1752.244} C_VEL
LIN {X 0,Y 583.735,Z 989.03,A -85,B 0,C 180,E1 1757.771,E2 1757.771} C_VEL
LIN {X 0,Y 583.746,Z 989.03,A -85,B 0,C 180,E1 1763.521,E2 1763.521} C_VEL
LIN {X 0,Y 583.676,Z 989.03,A -85,B 0,C 180,E1 1768.865,E2 1768.865} C_VEL
LIN {X 0,Y 583.837,Z 989.03,A -85,B 0,C 180,E1 1774.772,E2 1774.772} C_VEL
LIN {X 0,Y 583.911,Z 989.03,A -85,B 0,C 180,E1 1780.37,E2 1780.37} C_VEL
LIN {X 0,Y 583.655,Z 989.03,A -85,B 0,C 180,E1 1785.017,E2 1785.017} C_VEL
LIN {X 0,Y 583.934,Z 989.03,A -85,B 0,C 180,E1 1789.579,E2 1789.579} C_VEL
LIN {X 0,Y 584.166,Z 989.03,A -85,B 0,C 180,E1 1794.069,E2 1794.069} C_VEL
LIN {X 0,Y 583.907,Z 989.03,A -85,B 0,C 180,E1 1800,E2 1800} C_VEL
LIN {X 0,Y 583.943,Z 989.03,A -85,B 0,C 180,E1 1804.446,E2 1804.446} C_VEL
LIN {X 0,Y 583.972,Z 989.03,A -85,B 0,C 180,E1 1808.919,E2 1808.919} C_VEL
LIN {X 0,Y 583.992,Z 989.03,A -85,B 0,C 180,E1 1813.447,E2 1813.447} C_VEL
LIN {X 0,Y 583.941,Z 989.03,A -85,B 0,C 180,E1 1818.065,E2 1818.065} C_VEL
LIN {X 0,Y 583.837,Z 989.03,A -85,B 0,C 180,E1 1822.81,E2 1822.81} C_VEL
LIN {X 0,Y 583.715,Z 989.03,A -85,B 0,C 180,E1 1828.483,E2 1828.483} C_VEL
LIN {X 0,Y 583.728,Z 989.03,A -85,B 0,C 180,E1 1834.66,E2 1834.66} C_VEL
LIN {X 0,Y 583.589,Z 989.03,A -85,B 0,C 180,E1 1840.271,E2 1840.271} C_VEL
LIN {X 0,Y 583.733,Z 989.03,A -85,B 0,C 180,E1 1846.369,E2 1846.369} C_VEL
LIN {X 0,Y 583.707,Z 989.03,A -85,B 0,C 180,E1 1851.651,E2 1851.651} C_VEL
LIN {X 0,Y 583.579,Z 989.03,A -85,B 0,C 180,E1 1857.111,E2 1857.111} C_VEL
LIN {X 0,Y 583.94,Z 989.406,A -85,B 0,C 180,E1 1862.366,E2 1862.366} C_VEL
LIN {X 0,Y 586.464,Z 1001.763,A -85,B 0,C 180,E1 1863.142,E2 1863.142} C_VEL
LIN {X 0,Y 585.999,Z 1037.054,A -85,B 0,C 180,E1 1865.401,E2 1865.401} C_VEL
LIN {X 0,Y 585.342,Z 1069.334,A -85,B 0,C 180,E1 1868.131,E2 1868.131} C_VEL
LIN {X 0,Y 584.787,Z 1098.65,A -85,B 0,C 180,E1 1871.378,E2 1871.378} C_VEL
LIN {X 0,Y 584.357,Z 1122.333,A -85,B 0,C 180,E1 1874.844,E2 1874.844} C_VEL
LIN {X 0,Y 584.141,Z 1140.151,A -85,B 0,C 180,E1 1878.335,E2 1878.335} C_VEL
LIN {X 0,Y 584.096,Z 1153.836,A -85,B 0,C 180,E1 1882.205,E2 1882.205} C_VEL
LIN {X 0,Y 583.999,Z 1161.03,A -85,B 0,C 180,E1 1885.555,E2 1885.555} C_VEL
LIN {X 0,Y 584.032,Z 1164.117,A -85,B 0,C 180,E1 1888.52,E2 1888.52} C_VEL
LIN {X 0,Y 584.194,Z 1164.055,A -85,B 0,C 180,E1 1891.481,E2 1891.481} C_VEL
LIN {X 0,Y 584.177,Z 1159.674,A -85,B 0,C 180,E1 1895.188,E2 1895.188} C_VEL
LIN {X 0,Y 584.195,Z 1148.911,A -85,B 0,C 180,E1 1899.291,E2 1899.291} C_VEL
LIN {X 0,Y 584.305,Z 1133.217,A -85,B 0,C 180,E1 1903.061,E2 1903.061} C_VEL
LIN {X 0,Y 584.56,Z 1112.102,A -85,B 0,C 180,E1 1906.681,E2 1906.681} C_VEL
LIN {X 0,Y 585.004,Z 1086.309,A -85,B 0,C 180,E1 1910.003,E2 1910.003} C_VEL
LIN {X 0,Y 585.599,Z 1057.328,A -85,B 0,C 180,E1 1912.88,E2 1912.88} C_VEL
LIN {X 0,Y 586.311,Z 1023.721,A -85,B 0,C 180,E1 1915.437,E2 1915.437} C_VEL
LIN {X 0,Y 586.191,Z 996.473,A -85,B 0,C 180,E1 1917.072,E2 1917.072} C_VEL
LIN {X 0,Y 584.034,Z 989.03,A -85,B 0,C 180,E1 1917.624,E2 1917.624} C_VEL
LIN {X 0,Y 583.828,Z 989.03,A -85,B 0,C 180,E1 1924.202,E2 1924.202} C_VEL
LIN {X 0,Y 583.587,Z 989.03,A -85,B 0,C 180,E1 1930.274,E2 1930.274} C_VEL
LIN {X 0,Y 583.727,Z 989.03,A -85,B 0,C 180,E1 1936.373,E2 1936.373} C_VEL
LIN {X 0,Y 583.717,Z 989.03,A -85,B 0,C 180,E1 1941.654,E2 1941.654} C_VEL
LIN {X 0,Y 583.555,Z 989.03,A -85,B 0,C 180,E1 1947.111,E2 1947.111} C_VEL
LIN {X 0,Y 583.647,Z 989.03,A -85,B 0,C 180,E1 1952.266,E2 1952.266} C_VEL
LIN {X 0,Y 583.638,Z 989.03,A -85,B 0,C 180,E1 1957.182,E2 1957.182} C_VEL
LIN {X 0,Y 583.955,Z 989.03,A -85,B 0,C 180,E1 1961.936,E2 1961.936} C_VEL
LIN {X 0,Y 583.698,Z 989.03,A -85,B 0,C 180,E1 1968.064,E2 1968.064} C_VEL
LIN {X 0,Y 584.162,Z 989.03,A -85,B 0,C 180,E1 1974.069,E2 1974.069} C_VEL
LIN {X 0,Y 583.939,Z 989.03,A -85,B 0,C 180,E1 1980,E2 1980} C_VEL
LIN {X 0,Y 583.962,Z 989.03,A -85,B 0,C 180,E1 1984.446,E2 1984.446} C_VEL
LIN {X 0,Y 583.811,Z 989.03,A -85,B 0,C 180,E1 1985.862,E2 1985.862} C_VEL
LIN {X 0,Y 580.021,Z 989.03,A -85,B 0,C 180,E1 1987.541,E2 1987.541} C_VEL
LIN {X 0,Y 576.005,Z 989.03,A -85,B 0,C 180,E1 1989.241,E2 1989.241} C_VEL
LIN {X 0,Y 575.94,Z 989.03,A -85,B 0,C 180,E1 1994.201,E2 1994.201} C_VEL
LIN {X 0,Y 575.856,Z 989.03,A -85,B 0,C 180,E1 1999.916,E2 1999.916} C_VEL
LIN {X 0,Y 575.744,Z 989.03,A -85,B 0,C 180,E1 2004.793,E2 2004.793} C_VEL
LIN {X 0,Y 575.731,Z 989.03,A -85,B 0,C 180,E1 2010.123,E2 2010.123} C_VEL
LIN {X 0,Y 575.895,Z 989.03,A -85,B 0,C 180,E1 2015.2,E2 2015.2} C_VEL
LIN {X 0,Y 575.804,Z 989.03,A -85,B 0,C 180,E1 2020.931,E2 2020.931} C_VEL
LIN {X 0,Y 575.776,Z 989.03,A -85,B 0,C 180,E1 2027.206,E2 2027.206} C_VEL
LIN {X 0,Y 575.891,Z 989.03,A -85,B 0,C 180,E1 2032.938,E2 2032.938} C_VEL
LIN {X 0,Y 576.068,Z 989.044,A -85,B 0,C 180,E1 2038.35,E2 2038.35} C_VEL
LIN {X 0,Y 581.083,Z 1003.261,A -85,B 0,C 180,E1 2038.855,E2 2038.855} C_VEL
LIN {X 0,Y 580.906,Z 1077.32,A -85,B 0,C 180,E1 2040,E2 2040} C_VEL
LIN {X 0,Y 580.379,Z 1114.883,A -85,B 0,C 180,E1 2041.137,E2 2041.137} C_VEL
LIN {X 0,Y 579.574,Z 1150.921,A -85,B 0,C 180,E1 2042.795,E2 2042.795} C_VEL
LIN {X 0,Y 578.681,Z 1185.884,A -85,B 0,C 180,E1 2045.027,E2 2045.027} C_VEL
LIN {X 0,Y 577.84,Z 1217.656,A -85,B 0,C 180,E1 2047.715,E2 2047.715} C_VEL
LIN {X 0,Y 577.095,Z 1247.086,A -85,B 0,C 180,E1 2050.967,E2 2050.967} C_VEL
LIN {X 0,Y 576.554,Z 1272.072,A -85,B 0,C 180,E1 2054.632,E2 2054.632} C_VEL
LIN {X 0,Y 576.279,Z 1290.752,A -85,B 0,C 180,E1 2058.369,E2 2058.369} C_VEL
LIN {X 0,Y 576.203,Z 1303.716,A -85,B 0,C 180,E1 2062.097,E2 2062.097} C_VEL
LIN {X 0,Y 576.074,Z 1310.955,A -85,B 0,C 180,E1 2065.492,E2 2065.492} C_VEL
LIN {X 0,Y 576.127,Z 1314.086,A -85,B 0,C 180,E1 2068.499,E2 2068.499} C_VEL
LIN {X 0,Y 576.277,Z 1314.087,A -85,B 0,C 180,E1 2071.5,E2 2071.5} C_VEL
LIN {X 0,Y 576.249,Z 1308.864,A -85,B 0,C 180,E1 2075.701,E2 2075.701} C_VEL
LIN {X 0,Y 576.282,Z 1299.074,A -85,B 0,C 180,E1 2079.419,E2 2079.419} C_VEL
LIN {X 0,Y 576.455,Z 1283.451,A -85,B 0,C 180,E1 2083.241,E2 2083.241} C_VEL
LIN {X 0,Y 576.773,Z 1262.377,A -85,B 0,C 180,E1 2086.918,E2 2086.918} C_VEL
LIN {X 0,Y 577.378,Z 1236.874,A -85,B 0,C 180,E1 2090.26,E2 2090.26} C_VEL
LIN {X 0,Y 578.123,Z 1206.63,A -85,B 0,C 180,E1 2093.301,E2 2093.301} C_VEL
LIN {X 0,Y 579.061,Z 1172.553,A -85,B 0,C 180,E1 2095.904,E2 2095.904} C_VEL
LIN {X 0,Y 579.918,Z 1136.764,A -85,B 0,C 180,E1 2097.929,E2 2097.929} C_VEL
LIN {X 0,Y 580.606,Z 1099.381,A -85,B 0,C 180,E1 2099.403,E2 2099.403} C_VEL
LIN {X 0,Y 581.185,Z 1064.637,A -85,B 0,C 180,E1 2100.248,E2 2100.248} C_VEL
LIN {X 0,Y 580.554,Z 1000.147,A -85,B 0,C 180,E1 2101.22,E2 2101.22} C_VEL
LIN {X 0,Y 575.825,Z 989.03,A -85,B 0,C 180,E1 2101.693,E2 2101.693} C_VEL
LIN {X 0,Y 575.921,Z 989.03,A -85,B 0,C 180,E1 2108.185,E2 2108.185} C_VEL
LIN {X 0,Y 575.683,Z 989.03,A -85,B 0,C 180,E1 2112.962,E2 2112.962} C_VEL
LIN {X 0,Y 575.803,Z 989.03,A -85,B 0,C 180,E1 2119.069,E2 2119.069} C_VEL
LIN {X 0,Y 575.709,Z 989.03,A -85,B 0,C 180,E1 2124.787,E2 2124.787} C_VEL
LIN {X 0,Y 575.747,Z 989.03,A -85,B 0,C 180,E1 2130.135,E2 2130.135} C_VEL
LIN {X 0,Y 575.885,Z 989.03,A -85,B 0,C 180,E1 2135.214,E2 2135.214} C_VEL
LIN {X 0,Y 575.997,Z 989.03,A -85,B 0,C 180,E1 2140.584,E2 2140.584} C_VEL
LIN {X 0,Y 575.792,Z 989.03,A -85,B 0,C 180,E1 2144.807,E2 2144.807} C_VEL
LIN {X 0,Y 575.894,Z 989.03,A -85,B 0,C 180,E1 2150.955,E2 2150.955} C_VEL
LIN {X 0,Y 575.965,Z 989.03,A -85,B 0,C 180,E1 2155.492,E2 2155.492} C_VEL
LIN {X 0,Y 576.006,Z 989.03,A -85,B 0,C 180,E1 2160,E2 2160} C_VEL
LIN {X 0,Y 576.029,Z 989.03,A -85,B 0,C 180,E1 2164.507,E2 2164.507} C_VEL
LIN {X 0,Y 576.051,Z 989.03,A -85,B 0,C 180,E1 2169.043,E2 2169.043} C_VEL
LIN {X 0,Y 575.923,Z 989.03,A -85,B 0,C 180,E1 2174.199,E2 2174.199} C_VEL
LIN {X 0,Y 575.865,Z 989.03,A -85,B 0,C 180,E1 2179.916,E2 2179.916} C_VEL
LIN {X 0,Y 575.755,Z 989.03,A -85,B 0,C 180,E1 2184.792,E2 2184.792} C_VEL
LIN {X 0,Y 575.679,Z 989.03,A -85,B 0,C 180,E1 2190.116,E2 2190.116} C_VEL
LIN {X 0,Y 575.696,Z 989.03,A -85,B 0,C 180,E1 2195.214,E2 2195.214} C_VEL
LIN {X 0,Y 575.644,Z 989.03,A -85,B 0,C 180,E1 2200.945,E2 2200.945} C_VEL
LIN {X 0,Y 575.8,Z 989.03,A -85,B 0,C 180,E1 2207.203,E2 2207.203} C_VEL
LIN {X 0,Y 575.836,Z 989.03,A -85,B 0,C 180,E1 2212.935,E2 2212.935} C_VEL
LIN {X 0,Y 575.774,Z 989.03,A -85,B 0,C 180,E1 2218.388,E2 2218.388} C_VEL
LIN {X 0,Y 575.998,Z 989.054,A -85,B 0,C 180,E1 2221.934,E2 2221.934} C_VEL
LIN {X 0,Y 579.242,Z 1004.337,A -85,B 0,C 180,E1 2222.924,E2 2222.924} C_VEL
LIN {X 0,Y 578.581,Z 1040.677,A -85,B 0,C 180,E1 2225.336,E2 2225.336} C_VEL
LIN {X 0,Y 577.696,Z 1073.728,A -85,B 0,C 180,E1 2228.27,E2 2228.27} C_VEL
LIN {X 0,Y 577.043,Z 1101.669,A -85,B 0,C 180,E1 2231.527,E2 2231.527} C_VEL
LIN {X 0,Y 576.558,Z 1124.621,A -85,B 0,C 180,E1 2235.041,E2 2235.041} C_VEL
LIN {X 0,Y 576.265,Z 1140.918,A -85,B 0,C 180,E1 2238.365,E2 2238.365} C_VEL
LIN {X 0,Y 576.201,Z 1153.834,A -85,B 0,C 180,E1 2242.098,E2 2242.098} C_VEL
LIN {X 0,Y 576.1,Z 1161.029,A -85,B 0,C 180,E1 2245.494,E2 2245.494} C_VEL
LIN {X 0,Y 576.13,Z 1164.117,A -85,B 0,C 180,E1 2248.5,E2 2248.5} C_VEL
LIN {X 0,Y 576.289,Z 1164.056,A -85,B 0,C 180,E1 2251.501,E2 2251.501} C_VEL
LIN {X 0,Y 576.2,Z 1158.872,A -85,B 0,C 180,E1 2255.652,E2 2255.652} C_VEL
LIN {X 0,Y 576.287,Z 1148.913,A -85,B 0,C 180,E1 2259.42,E2 2259.42} C_VEL
LIN {X 0,Y 576.441,Z 1133.219,A -85,B 0,C 180,E1 2263.242,E2 2263.242} C_VEL
LIN {X 0,Y 576.787,Z 1112.107,A -85,B 0,C 180,E1 2266.912,E2 2266.912} C_VEL
LIN {X 0,Y 577.336,Z 1086.469,A -85,B 0,C 180,E1 2270.263,E2 2270.263} C_VEL
LIN {X 0,Y 578.155,Z 1056.088,A -85,B 0,C 180,E1 2273.303,E2 2273.303} C_VEL
LIN {X 0,Y 579.046,Z 1022.963,A -85,B 0,C 180,E1 2275.832,E2 2275.832} C_VEL
LIN {X 0,Y 578.682,Z 998.284,A -85,B 0,C 180,E1 2277.353,E2 2277.353} C_VEL
LIN {X 0,Y 576.037,Z 989.03,A -85,B 0,C 180,E1 2278,E2 2278} C_VEL
LIN {X 0,Y 575.884,Z 989.03,A -85,B 0,C 180,E1 2283.386,E2 2283.386} C_VEL
LIN {X 0,Y 575.679,Z 989.03,A -85,B 0,C 180,E1 2288.985,E2 2288.985} C_VEL
LIN {X 0,Y 575.742,Z 989.03,A -85,B 0,C 180,E1 2295.046,E2 2295.046} C_VEL
LIN {X 0,Y 575.756,Z 989.03,A -85,B 0,C 180,E1 2301.024,E2 2301.024} C_VEL
LIN {X 0,Y 575.659,Z 989.03,A -85,B 0,C 180,E1 2306.601,E2 2306.601} C_VEL
LIN {X 0,Y 575.728,Z 989.03,A -85,B 0,C 180,E1 2311.851,E2 2311.851} C_VEL
LIN {X 0,Y 575.726,Z 989.03,A -85,B 0,C 180,E1 2316.85,E2 2316.85} C_VEL
LIN {X 0,Y 576.025,Z 989.03,A -85,B 0,C 180,E1 2321.678,E2 2321.678} C_VEL
LIN {X 0,Y 575.755,Z 989.03,A -85,B 0,C 180,E1 2327.897,E2 2327.897} C_VEL
LIN {X 0,Y 576.246,Z 989.03,A -85,B 0,C 180,E1 2333.988,E2 2333.988} C_VEL
LIN {X 0,Y 576.038,Z 989.03,A -85,B 0,C 180,E1 2340,E2 2340} C_VEL
LIN {X 0,Y 575.932,Z 989.03,A -85,B 0,C 180,E1 2345.342,E2 2345.342} C_VEL
LIN {X 0,Y 576.005,Z 989.03,A -85,B 0,C 180,E1 2349.241,E2 2349.241} C_VEL
LIN {X 0,Y 571.949,Z 989.03,A -85,B 0,C 180,E1 2350.936,E2 2350.936} C_VEL
LIN {X 0,Y 568.047,Z 989.03,A -85,B 0,C 180,E1 2352.654,E2 2352.654} C_VEL
LIN {X 0,Y 568.055,Z 989.03,A -85,B 0,C 180,E1 2358.588,E2 2358.588} C_VEL
LIN {X 0,Y 567.941,Z 989.03,A -85,B 0,C 180,E1 2363.486,E2 2363.486} C_VEL
LIN {X 0,Y 567.874,Z 989.03,A -85,B 0,C 180,E1 2368.727,E2 2368.727} C_VEL
LIN {X 0,Y 567.974,Z 989.03,A -85,B 0,C 180,E1 2374.55,E2 2374.55} C_VEL
LIN {X 0,Y 567.83,Z 989.03,A -85,B 0,C 180,E1 2379.626,E2 2379.626} C_VEL
LIN {X 0,Y 567.68,Z 989.03,A -85,B 0,C 180,E1 2384.133,E2 2384.133} C_VEL
LIN {X 0,Y 567.829,Z 989.03,A -85,B 0,C 180,E1 2388.365,E2 2388.365} C_VEL
LIN {X 0,Y 568.006,Z 989.03,A -85,B 0,C 180,E1 2394.234,E2 2394.234} C_VEL
LIN {X 0,Y 568.138,Z 989.049,A -85,B 0,C 180,E1 2397.856,E2 2397.856} C_VEL
LIN {X 0,Y 574.267,Z 1003.843,A -85,B 0,C 180,E1 2398.452,E2 2398.452} C_VEL
LIN {X 0,Y 574.051,Z 1077.321,A -85,B 0,C 180,E1 2399.604,E2 2399.604} C_VEL
LIN {X 0,Y 573.386,Z 1114.675,A -85,B 0,C 180,E1 2400.743,E2 2400.743} C_VEL
LIN {X 0,Y 572.398,Z 1150.828,A -85,B 0,C 180,E1 2402.42,E2 2402.42} C_VEL
LIN {X 0,Y 571.342,Z 1186.1,A -85,B 0,C 180,E1 2404.7,E2 2404.7} C_VEL
LIN {X 0,Y 570.3,Z 1218.607,A -85,B 0,C 180,E1 2407.498,E2 2407.498} C_VEL
LIN {X 0,Y 569.419,Z 1247.67,A -85,B 0,C 180,E1 2410.775,E2 2410.775} C_VEL
LIN {X 0,Y 568.723,Z 1272.073,A -85,B 0,C 180,E1 2414.415,E2 2414.415} C_VEL
LIN {X 0,Y 568.421,Z 1290.441,A -85,B 0,C 180,E1 2418.127,E2 2418.127} C_VEL
LIN {X 0,Y 568.318,Z 1303.716,A -85,B 0,C 180,E1 2421.986,E2 2421.986} C_VEL
LIN {X 0,Y 568.195,Z 1310.955,A -85,B 0,C 180,E1 2425.43,E2 2425.43} C_VEL
LIN {X 0,Y 568.256,Z 1314.086,A -85,B 0,C 180,E1 2428.478,E2 2428.478} C_VEL
LIN {X 0,Y 568.393,Z 1314.087,A -85,B 0,C 180,E1 2431.521,E2 2431.521} C_VEL
LIN {X 0,Y 568.359,Z 1309.363,A -85,B 0,C 180,E1 2435.534,E2 2435.534} C_VEL
LIN {X 0,Y 568.371,Z 1299.074,A -85,B 0,C 180,E1 2439.551,E2 2439.551} C_VEL
LIN {X 0,Y 568.599,Z 1283.449,A -85,B 0,C 180,E1 2443.427,E2 2443.427} C_VEL
LIN {X 0,Y 569.031,Z 1262.105,A -85,B 0,C 180,E1 2447.196,E2 2447.196} C_VEL
LIN {X 0,Y 569.764,Z 1236.873,A -85,B 0,C 180,E1 2450.543,E2 2450.543} C_VEL
LIN {X 0,Y 570.639,Z 1207.124,A -85,B 0,C 180,E1 2453.58,E2 2453.58} C_VEL
LIN {X 0,Y 571.763,Z 1173.49,A -85,B 0,C 180,E1 2456.195,E2 2456.195} C_VEL
LIN {X 0,Y 572.791,Z 1138.331,A -85,B 0,C 180,E1 2458.228,E2 2458.228} C_VEL
LIN {X 0,Y 573.636,Z 1102.216,A -85,B 0,C 180,E1 2459.701,E2 2459.701} C_VEL
LIN {X 0,Y 574.354,Z 1064.637,A -85,B 0,C 180,E1 2460.646,E2 2460.646} C_VEL
LIN {X 0,Y 573.8,Z 1002.7,A -85,B 0,C 180,E1 2461.593,E2 2461.593} C_VEL
LIN {X 0,Y 567.778,Z 989.03,A -85,B 0,C 180,E1 2462.22,E2 2462.22} C_VEL
LIN {X 0,Y 568.004,Z 989.03,A -85,B 0,C 180,E1 2467.664,E2 2467.664} C_VEL
LIN {X 0,Y 567.741,Z 989.03,A -85,B 0,C 180,E1 2474.143,E2 2474.143} C_VEL
LIN {X 0,Y 567.832,Z 989.03,A -85,B 0,C 180,E1 2478.368,E2 2478.368} C_VEL
LIN {X 0,Y 567.848,Z 989.03,A -85,B 0,C 180,E1 2484.225,E2 2484.225} C_VEL
LIN {X 0,Y 567.84,Z 989.03,A -85,B 0,C 180,E1 2489.676,E2 2489.676} C_VEL
LIN {X 0,Y 567.933,Z 989.03,A -85,B 0,C 180,E1 2494.843,E2 2494.843} C_VEL
LIN {X 0,Y 568.012,Z 989.03,A -85,B 0,C 180,E1 2499.797,E2 2499.797} C_VEL
LIN {X 0,Y 567.9,Z 989.03,A -85,B 0,C 180,E1 2504.591,E2 2504.591} C_VEL
LIN {X 0,Y 567.988,Z 989.03,A -85,B 0,C 180,E1 2510.828,E2 2510.828} C_VEL
LIN {X 0,Y 568.074,Z 989.03,A -85,B 0,C 180,E1 2515.429,E2 2515.429} C_VEL
LIN {X 0,Y 568.131,Z 989.03,A -85,B 0,C 180,E1 2520,E2 2520} C_VEL
LIN {X 0,Y 568.116,Z 989.03,A -85,B 0,C 180,E1 2524.57,E2 2524.57} C_VEL
LIN {X 0,Y 568.118,Z 989.03,A -85,B 0,C 180,E1 2529.17,E2 2529.17} C_VEL
LIN {X 0,Y 568.11,Z 989.03,A -85,B 0,C 180,E1 2533.83,E2 2533.83} C_VEL
LIN {X 0,Y 568.062,Z 989.03,A -85,B 0,C 180,E1 2538.588,E2 2538.588} C_VEL
LIN {X 0,Y 567.952,Z 989.03,A -85,B 0,C 180,E1 2543.486,E2 2543.486} C_VEL
LIN {X 0,Y 567.845,Z 989.03,A -85,B 0,C 180,E1 2548.724,E2 2548.724} C_VEL
LIN {X 0,Y 567.798,Z 989.03,A -85,B 0,C 180,E1 2554.526,E2 2554.526} C_VEL
LIN {X 0,Y 567.745,Z 989.03,A -85,B 0,C 180,E1 2559.633,E2 2559.633} C_VEL
LIN {X 0,Y 567.786,Z 989.03,A -85,B 0,C 180,E1 2565.853,E2 2565.853} C_VEL
LIN {X 0,Y 567.844,Z 989.03,A -85,B 0,C 180,E1 2570.41,E2 2570.41} C_VEL
LIN {X 0,Y 567.728,Z 989.03,A -85,B 0,C 180,E1 2575.481,E2 2575.481} C_VEL
LIN {X 0,Y 568.024,Z 989.4,A -85,B 0,C 180,E1 2581.523,E2 2581.523} C_VEL
LIN {X 0,Y 572.045,Z 1006.1,A -85,B 0,C 180,E1 2582.655,E2 2582.655} C_VEL
LIN {X 0,Y 571.109,Z 1043.163,A -85,B 0,C 180,E1 2585.196,E2 2585.196} C_VEL
LIN {X 0,Y 570.097,Z 1075.316,A -85,B 0,C 180,E1 2588.136,E2 2588.136} C_VEL
LIN {X 0,Y 569.302,Z 1103.037,A -85,B 0,C 180,E1 2591.454,E2 2591.454} C_VEL
LIN {X 0,Y 568.736,Z 1125.458,A -85,B 0,C 180,E1 2594.981,E2 2594.981} C_VEL
LIN {X 0,Y 568.422,Z 1142.468,A -85,B 0,C 180,E1 2598.593,E2 2598.593} C_VEL
LIN {X 0,Y 568.315,Z 1154.792,A -85,B 0,C 180,E1 2602.371,E2 2602.371} C_VEL
LIN {X 0,Y 568.22,Z 1161.029,A -85,B 0,C 180,E1 2605.431,E2 2605.431} C_VEL
LIN {X 0,Y 568.258,Z 1164.117,A -85,B 0,C 180,E1 2608.479,E2 2608.479} C_VEL
LIN {X 0,Y 568.404,Z 1164.057,A -85,B 0,C 180,E1 2611.522,E2 2611.522} C_VEL
LIN {X 0,Y 568.317,Z 1159.369,A -85,B 0,C 180,E1 2615.487,E2 2615.487} C_VEL
LIN {X 0,Y 568.377,Z 1148.915,A -85,B 0,C 180,E1 2619.552,E2 2619.552} C_VEL
LIN {X 0,Y 568.589,Z 1133.221,A -85,B 0,C 180,E1 2623.428,E2 2623.428} C_VEL
LIN {X 0,Y 569.026,Z 1111.863,A -85,B 0,C 180,E1 2627.187,E2 2627.187} C_VEL
LIN {X 0,Y 569.758,Z 1086.476,A -85,B 0,C 180,E1 2630.545,E2 2630.545} C_VEL
LIN {X 0,Y 570.701,Z 1056.6,A -85,B 0,C 180,E1 2633.58,E2 2633.58} C_VEL
LIN {X 0,Y 571.781,Z 1022.777,A -85,B 0,C 180,E1 2636.199,E2 2636.199} C_VEL
LIN {X 0,Y 571.926,Z 1002.163,A -85,B 0,C 180,E1 2637.484,E2 2637.484} C_VEL
LIN {X 0,Y 568.018,Z 989.03,A -85,B 0,C 180,E1 2638.451,E2 2638.451} C_VEL
LIN {X 0,Y 567.801,Z 989.03,A -85,B 0,C 180,E1 2644.53,E2 2644.53} C_VEL
LIN {X 0,Y 567.749,Z 989.03,A -85,B 0,C 180,E1 2649.636,E2 2649.636} C_VEL
LIN {X 0,Y 567.782,Z 989.03,A -85,B 0,C 180,E1 2655.857,E2 2655.857} C_VEL
LIN {X 0,Y 567.854,Z 989.03,A -85,B 0,C 180,E1 2660.413,E2 2660.413} C_VEL
LIN {X 0,Y 567.721,Z 989.03,A -85,B 0,C 180,E1 2665.487,E2 2665.487} C_VEL
LIN {X 0,Y 567.836,Z 989.03,A -85,B 0,C 180,E1 2669.675,E2 2669.675} C_VEL
LIN {X 0,Y 567.934,Z 989.03,A -85,B 0,C 180,E1 2674.843,E2 2674.843} C_VEL
LIN {X 0,Y 568.062,Z 989.03,A -85,B 0,C 180,E1 2679.799,E2 2679.799} C_VEL
LIN {X 0,Y 567.891,Z 989.03,A -85,B 0,C 180,E1 2684.591,E2 2684.591} C_VEL
LIN {X 0,Y 567.997,Z 989.03,A -85,B 0,C 180,E1 2690.828,E2 2690.828} C_VEL
LIN {X 0,Y 568.087,Z 989.03,A -85,B 0,C 180,E1 2695.43,E2 2695.43} C_VEL
LIN {X 0,Y 568.162,Z 989.03,A -85,B 0,C 180,E1 2700,E2 2700} C_VEL
LIN {X 0,Y 568.134,Z 989.03,A -85,B 0,C 180,E1 2704.57,E2 2704.57} C_VEL
LIN {X 0,Y 568.108,Z 989.03,A -85,B 0,C 180,E1 2709.224,E2 2709.224} C_VEL
LIN {X 0,Y 568.047,Z 989.03,A -85,B 0,C 180,E1 2712.654,E2 2712.654} C_VEL
LIN {X 0,Y 566.755,Z 989.03,A -85,B 0,C 180,E1 2713.525,E2 2713.525} C_VEL
LIN {X 0,Y 560.081,Z 989.03,A -85,B 0,C 180,E1 2715.895,E2 2715.895} C_VEL
LIN {X 0,Y 559.992,Z 989.03,A -85,B 0,C 180,E1 2716.119,E2 2716.119} C_VEL
LIN {X 0,Y 560.008,Z 989.03,A -85,B 0,C 180,E1 2720.505,E2 2720.505} C_VEL
LIN {X 0,Y 559.885,Z 989.03,A -85,B 0,C 180,E1 2725.545,E2 2725.545} C_VEL
LIN {X 0,Y 559.938,Z 989.03,A -85,B 0,C 180,E1 2730.798,E2 2730.798} C_VEL
LIN {X 0,Y 560.041,Z 989.03,A -85,B 0,C 180,E1 2736.353,E2 2736.353} C_VEL
LIN {X 0,Y 559.854,Z 989.03,A -85,B 0,C 180,E1 2742.362,E2 2742.362} C_VEL
LIN {X 0,Y 559.866,Z 989.03,A -85,B 0,C 180,E1 2747.636,E2 2747.636} C_VEL
LIN {X 0,Y 560.106,Z 989.03,A -85,B 0,C 180,E1 2753.922,E2 2753.922} C_VEL
LIN {X 0,Y 560.261,Z 989.094,A -85,B 0,C 180,E1 2757.349,E2 2757.349} C_VEL
LIN {X 0,Y 567.591,Z 1008.048,A -85,B 0,C 180,E1 2758.099,E2 2758.099} C_VEL
LIN {X 0,Y 567.221,Z 1079.237,A -85,B 0,C 180,E1 2759.242,E2 2759.242} C_VEL
LIN {X 0,Y 566.36,Z 1118.335,A -85,B 0,C 180,E1 2760.489,E2 2760.489} C_VEL
LIN {X 0,Y 565.164,Z 1156.394,A -85,B 0,C 180,E1 2762.357,E2 2762.357} C_VEL
LIN {X 0,Y 563.808,Z 1191.835,A -85,B 0,C 180,E1 2764.787,E2 2764.787} C_VEL
LIN {X 0,Y 562.604,Z 1224.081,A -85,B 0,C 180,E1 2767.742,E2 2767.742} C_VEL
LIN {X 0,Y 561.621,Z 1251.668,A -85,B 0,C 180,E1 2771.046,E2 2771.046} C_VEL
LIN {X 0,Y 560.923,Z 1273.166,A -85,B 0,C 180,E1 2774.393,E2 2774.393} C_VEL
LIN {X 0,Y 560.568,Z 1290.44,A -85,B 0,C 180,E1 2777.958,E2 2777.958} C_VEL
LIN {X 0,Y 560.456,Z 1303.716,A -85,B 0,C 180,E1 2781.873,E2 2781.873} C_VEL
LIN {X 0,Y 560.317,Z 1310.956,A -85,B 0,C 180,E1 2785.365,E2 2785.365} C_VEL
LIN {X 0,Y 560.355,Z 1314.086,A -85,B 0,C 180,E1 2788.456,E2 2788.456} C_VEL
LIN {X 0,Y 560.486,Z 1314.087,A -85,B 0,C 180,E1 2791.542,E2 2791.542} C_VEL
LIN {X 0,Y 560.479,Z 1309.825,A -85,B 0,C 180,E1 2795.364,E2 2795.364} C_VEL
LIN {X 0,Y 560.515,Z 1300.304,A -85,B 0,C 180,E1 2799.295,E2 2799.295} C_VEL
LIN {X 0,Y 560.773,Z 1285.283,A -85,B 0,C 180,E1 2803.222,E2 2803.222} C_VEL
LIN {X 0,Y 561.215,Z 1264.922,A -85,B 0,C 180,E1 2807.002,E2 2807.002} C_VEL
LIN {X 0,Y 562.084,Z 1238.619,A -85,B 0,C 180,E1 2810.631,E2 2810.631} C_VEL
LIN {X 0,Y 563.194,Z 1207.985,A -85,B 0,C 180,E1 2813.832,E2 2813.832} C_VEL
LIN {X 0,Y 564.449,Z 1174.956,A -85,B 0,C 180,E1 2816.457,E2 2816.457} C_VEL
LIN {X 0,Y 565.681,Z 1140.159,A -85,B 0,C 180,E1 2818.521,E2 2818.521} C_VEL
LIN {X 0,Y 566.705,Z 1103.293,A -85,B 0,C 180,E1 2820.065,E2 2820.065} C_VEL
LIN {X 0,Y 567.554,Z 1066.067,A -85,B 0,C 180,E1 2821.029,E2 2821.029} C_VEL
LIN {X 0,Y 566.92,Z 1005.146,A -85,B 0,C 180,E1 2821.986,E2 2821.986} C_VEL
LIN {X 0,Y 559.832,Z 989.03,A -85,B 0,C 180,E1 2822.708,E2 2822.708} C_VEL
LIN {X 0,Y 559.995,Z 989.03,A -85,B 0,C 180,E1 2828.299,E2 2828.299} C_VEL
LIN {X 0,Y 559.811,Z 989.03,A -85,B 0,C 180,E1 2834.494,E2 2834.494} C_VEL
LIN {X 0,Y 559.849,Z 989.03,A -85,B 0,C 180,E1 2839.694,E2 2839.694} C_VEL
LIN {X 0,Y 559.842,Z 989.03,A -85,B 0,C 180,E1 2845.527,E2 2845.527} C_VEL
LIN {X 0,Y 559.873,Z 989.03,A -85,B 0,C 180,E1 2850.979,E2 2850.979} C_VEL
LIN {X 0,Y 559.953,Z 989.03,A -85,B 0,C 180,E1 2856.385,E2 2856.385} C_VEL
LIN {X 0,Y 560.128,Z 989.03,A -85,B 0,C 180,E1 2861.139,E2 2861.139} C_VEL
LIN {X 0,Y 559.85,Z 989.03,A -85,B 0,C 180,E1 2866.008,E2 2866.008} C_VEL
LIN {X 0,Y 560.081,Z 989.03,A -85,B 0,C 180,E1 2870.697,E2 2870.697} C_VEL
LIN {X 0,Y 560.184,Z 989.03,A -85,B 0,C 180,E1 2875.365,E2 2875.365} C_VEL
LIN {X 0,Y 560.23,Z 989.03,A -85,B 0,C 180,E1 2880,E2 2880} C_VEL
LIN {X 0,Y 560.195,Z 989.03,A -85,B 0,C 180,E1 2884.677,E2 2884.677} C_VEL
LIN {X 0,Y 560.22,Z 989.03,A -85,B 0,C 180,E1 2889.3,E2 2889.3} C_VEL
LIN {X 0,Y 560.142,Z 989.03,A -85,B 0,C 180,E1 2894.111,E2 2894.111} C_VEL
LIN {X 0,Y 560.053,Z 989.03,A -85,B 0,C 180,E1 2899.432,E2 2899.432} C_VEL
LIN {X 0,Y 559.988,Z 989.03,A -85,B 0,C 180,E1 2903.84,E2 2903.84} C_VEL
LIN {X 0,Y 559.906,Z 989.03,A -85,B 0,C 180,E1 2909.019,E2 2909.019} C_VEL
LIN {X 0,Y 559.916,Z 989.03,A -85,B 0,C 180,E1 2914.467,E2 2914.467} C_VEL
LIN {X 0,Y 559.755,Z 989.03,A -85,B 0,C 180,E1 2920.99,E2 2920.99} C_VEL
LIN {X 0,Y 559.857,Z 989.03,A -85,B 0,C 180,E1 2926.695,E2 2926.695} C_VEL
LIN {X 0,Y 559.913,Z 989.03,A -85,B 0,C 180,E1 2931.694,E2 2931.694} C_VEL
LIN {X 0,Y 559.828,Z 989.03,A -85,B 0,C 180,E1 2937.378,E2 2937.378} C_VEL
LIN {X 0,Y 560.127,Z 989.742,A -85,B 0,C 180,E1 2941.102,E2 2941.102} C_VEL
LIN {X 0,Y 564.85,Z 1008.37,A -85,B 0,C 180,E1 2942.419,E2 2942.419} C_VEL
LIN {X 0,Y 563.699,Z 1044.098,A -85,B 0,C 180,E1 2944.926,E2 2944.926} C_VEL
LIN {X 0,Y 562.556,Z 1074.573,A -85,B 0,C 180,E1 2947.748,E2 2947.748} C_VEL
LIN {X 0,Y 561.583,Z 1102.013,A -85,B 0,C 180,E1 2951.048,E2 2951.048} C_VEL
LIN {X 0,Y 560.921,Z 1123.418,A -85,B 0,C 180,E1 2954.394,E2 2954.394} C_VEL
LIN {X 0,Y 560.549,Z 1140.62,A -85,B 0,C 180,E1 2957.958,E2 2957.958} C_VEL
LIN {X 0,Y 560.455,Z 1153.831,A -85,B 0,C 180,E1 2961.874,E2 2961.874} C_VEL
LIN {X 0,Y 560.339,Z 1161.028,A -85,B 0,C 180,E1 2965.367,E2 2965.367} C_VEL
LIN {X 0,Y 560.355,Z 1164.117,A -85,B 0,C 180,E1 2968.457,E2 2968.457} C_VEL
LIN {X 0,Y 560.498,Z 1164.057,A -85,B 0,C 180,E1 2971.543,E2 2971.543} C_VEL
LIN {X 0,Y 560.427,Z 1159.747,A -85,B 0,C 180,E1 2975.368,E2 2975.368} C_VEL
LIN {X 0,Y 560.52,Z 1150.169,A -85,B 0,C 180,E1 2979.296,E2 2979.296} C_VEL
LIN {X 0,Y 560.762,Z 1135.081,A -85,B 0,C 180,E1 2983.223,E2 2983.223} C_VEL
LIN {X 0,Y 561.25,Z 1113.371,A -85,B 0,C 180,E1 2987.203,E2 2987.203} C_VEL
LIN {X 0,Y 562.08,Z 1088.227,A -85,B 0,C 180,E1 2990.633,E2 2990.633} C_VEL
LIN {X 0,Y 563.176,Z 1058.951,A -85,B 0,C 180,E1 2993.699,E2 2993.699} C_VEL
LIN {X 0,Y 564.423,Z 1025.697,A -85,B 0,C 180,E1 2996.362,E2 2996.362} C_VEL
LIN {X 0,Y 564.708,Z 1004.471,A -85,B 0,C 180,E1 2997.734,E2 2997.734} C_VEL
LIN {X 0,Y 560.02,Z 989.03,A -85,B 0,C 180,E1 2998.852,E2 2998.852} C_VEL
LIN {X 0,Y 559.919,Z 989.03,A -85,B 0,C 180,E1 3004.47,E2 3004.47} C_VEL
LIN {X 0,Y 559.748,Z 989.03,A -85,B 0,C 180,E1 3010.317,E2 3010.317} C_VEL
LIN {X 0,Y 559.831,Z 989.03,A -85,B 0,C 180,E1 3015.509,E2 3015.509} C_VEL
LIN {X 0,Y 559.905,Z 989.03,A -85,B 0,C 180,E1 3021.407,E2 3021.407} C_VEL
LIN {X 0,Y 559.796,Z 989.03,A -85,B 0,C 180,E1 3026.685,E2 3026.685} C_VEL
LIN {X 0,Y 559.873,Z 989.03,A -85,B 0,C 180,E1 3030.979,E2 3030.979} C_VEL
LIN {X 0,Y 559.937,Z 989.03,A -85,B 0,C 180,E1 3036.391,E2 3036.391} C_VEL
LIN {X 0,Y 560.183,Z 989.03,A -85,B 0,C 180,E1 3041.141,E2 3041.141} C_VEL
LIN {X 0,Y 559.831,Z 989.03,A -85,B 0,C 180,E1 3046.021,E2 3046.021} C_VEL
LIN {X 0,Y 560.091,Z 989.03,A -85,B 0,C 180,E1 3050.698,E2 3050.698} C_VEL
LIN {X 0,Y 560.195,Z 989.03,A -85,B 0,C 180,E1 3055.365,E2 3055.365} C_VEL
LIN {X 0,Y 560.26,Z 989.03,A -85,B 0,C 180,E1 3060,E2 3060} C_VEL
LIN {X 0,Y 560.234,Z 989.03,A -85,B 0,C 180,E1 3064.713,E2 3064.713} C_VEL
LIN {X 0,Y 560.203,Z 989.03,A -85,B 0,C 180,E1 3069.301,E2 3069.301} C_VEL
LIN {X 0,Y 560.173,Z 989.03,A -85,B 0,C 180,E1 3074.12,E2 3074.12} C_VEL
LIN {X 0,Y 559.992,Z 989.03,A -85,B 0,C 180,E1 3076.119,E2 3076.119} C_VEL
LIN {X 0,Y 558.774,Z 989.03,A -85,B 0,C 180,E1 3077.003,E2 3077.003} C_VEL
LIN {X 0,Y 552.1,Z 989.03,A -85,B 0,C 180,E1 3079.635,E2 3079.635} C_VEL
LIN {X 0,Y 551.988,Z 989.03,A -85,B 0,C 180,E1 3085.557,E2 3085.557} C_VEL
LIN {X 0,Y 552.007,Z 989.03,A -85,B 0,C 180,E1 3091.29,E2 3091.29} C_VEL
LIN {X 0,Y 552.034,Z 989.03,A -85,B 0,C 180,E1 3096.967,E2 3096.967} C_VEL
LIN {X 0,Y 551.906,Z 989.03,A -85,B 0,C 180,E1 3103.119,E2 3103.119} C_VEL
LIN {X 0,Y 552,Z 989.03,A -85,B 0,C 180,E1 3108.997,E2 3108.997} C_VEL
LIN {X 0,Y 552.169,Z 989.03,A -85,B 0,C 180,E1 3115.068,E2 3115.068} C_VEL
LIN {X 0,Y 552.324,Z 989.107,A -85,B 0,C 180,E1 3116.82,E2 3116.82} C_VEL
LIN {X 0,Y 560.888,Z 1009.533,A -85,B 0,C 180,E1 3117.693,E2 3117.693} C_VEL
LIN {X 0,Y 560.41,Z 1079.238,A -85,B 0,C 180,E1 3118.827,E2 3118.827} C_VEL
LIN {X 0,Y 559.429,Z 1118.208,A -85,B 0,C 180,E1 3120.081,E2 3120.081} C_VEL
LIN {X 0,Y 558.032,Z 1156.19,A -85,B 0,C 180,E1 3121.96,E2 3121.96} C_VEL
LIN {X 0,Y 556.431,Z 1192.966,A -85,B 0,C 180,E1 3124.525,E2 3124.525} C_VEL
LIN {X 0,Y 555.086,Z 1224.227,A -85,B 0,C 180,E1 3127.44,E2 3127.44} C_VEL
LIN {X 0,Y 553.928,Z 1250.901,A -85,B 0,C 180,E1 3130.664,E2 3130.664} C_VEL
LIN {X 0,Y 553.094,Z 1273.167,A -85,B 0,C 180,E1 3134.167,E2 3134.167} C_VEL
LIN {X 0,Y 552.725,Z 1290.441,A -85,B 0,C 180,E1 3137.784,E2 3137.784} C_VEL
LIN {X 0,Y 552.592,Z 1303.716,A -85,B 0,C 180,E1 3141.757,E2 3141.757} C_VEL
LIN {X 0,Y 552.44,Z 1310.956,A -85,B 0,C 180,E1 3145.299,E2 3145.299} C_VEL
LIN {X 0,Y 552.46,Z 1314.087,A -85,B 0,C 180,E1 3148.434,E2 3148.434} C_VEL
LIN {X 0,Y 552.58,Z 1314.088,A -85,B 0,C 180,E1 3151.564,E2 3151.564} C_VEL
LIN {X 0,Y 552.541,Z 1309.378,A -85,B 0,C 180,E1 3155.686,E2 3155.686} C_VEL
LIN {X 0,Y 552.616,Z 1300.304,A -85,B 0,C 180,E1 3159.429,E2 3159.429} C_VEL
LIN {X 0,Y 552.921,Z 1285.284,A -85,B 0,C 180,E1 3163.413,E2 3163.413} C_VEL
LIN {X 0,Y 553.512,Z 1263.671,A -85,B 0,C 180,E1 3167.45,E2 3167.45} C_VEL
LIN {X 0,Y 554.473,Z 1238.618,A -85,B 0,C 180,E1 3170.928,E2 3170.928} C_VEL
LIN {X 0,Y 555.768,Z 1207.986,A -85,B 0,C 180,E1 3174.171,E2 3174.171} C_VEL
LIN {X 0,Y 557.174,Z 1175.676,A -85,B 0,C 180,E1 3176.779,E2 3176.779} C_VEL
LIN {X 0,Y 558.626,Z 1140.646,A -85,B 0,C 180,E1 3178.89,E2 3178.89} C_VEL
LIN {X 0,Y 559.835,Z 1103.761,A -85,B 0,C 180,E1 3180.457,E2 3180.457} C_VEL
LIN {X 0,Y 560.78,Z 1066.067,A -85,B 0,C 180,E1 3181.446,E2 3181.446} C_VEL
LIN {X 0,Y 560.455,Z 1008.093,A -85,B 0,C 180,E1 3182.356,E2 3182.356} C_VEL
LIN {X 0,Y 551.912,Z 989.03,A -85,B 0,C 180,E1 3183.259,E2 3183.259} C_VEL
LIN {X 0,Y 552.024,Z 989.03,A -85,B 0,C 180,E1 3188.956,E2 3188.956} C_VEL
LIN {X 0,Y 551.929,Z 989.03,A -85,B 0,C 180,E1 3195.304,E2 3195.304} C_VEL
LIN {X 0,Y 551.962,Z 989.03,A -85,B 0,C 180,E1 3201.041,E2 3201.041} C_VEL
LIN {X 0,Y 551.896,Z 989.03,A -85,B 0,C 180,E1 3206.851,E2 3206.851} C_VEL
LIN {X 0,Y 551.978,Z 989.03,A -85,B 0,C 180,E1 3212.307,E2 3212.307} C_VEL
LIN {X 0,Y 552.023,Z 989.03,A -85,B 0,C 180,E1 3217.5,E2 3217.5} C_VEL
LIN {X 0,Y 552.227,Z 989.03,A -85,B 0,C 180,E1 3223.019,E2 3223.019} C_VEL
LIN {X 0,Y 552.185,Z 989.03,A -85,B 0,C 180,E1 3229.672,E2 3229.672} C_VEL
LIN {X 0,Y 552.319,Z 989.03,A -85,B 0,C 180,E1 3235.299,E2 3235.299} C_VEL
LIN {X 0,Y 552.333,Z 989.03,A -85,B 0,C 180,E1 3240,E2 3240} C_VEL
LIN {X 0,Y 552.318,Z 989.03,A -85,B 0,C 180,E1 3244.701,E2 3244.701} C_VEL
LIN {X 0,Y 552.177,Z 989.03,A -85,B 0,C 180,E1 3250.323,E2 3250.323} C_VEL
LIN {X 0,Y 552.1,Z 989.03,A -85,B 0,C 180,E1 3255.861,E2 3255.861} C_VEL
LIN {X 0,Y 552.077,Z 989.03,A -85,B 0,C 180,E1 3261.67,E2 3261.67} C_VEL
LIN {X 0,Y 551.985,Z 989.03,A -85,B 0,C 180,E1 3267.692,E2 3267.692} C_VEL
LIN {X 0,Y 552.037,Z 989.03,A -85,B 0,C 180,E1 3273.14,E2 3273.14} C_VEL
LIN {X 0,Y 551.823,Z 989.03,A -85,B 0,C 180,E1 3278.971,E2 3278.971} C_VEL
LIN {X 0,Y 551.905,Z 989.03,A -85,B 0,C 180,E1 3284.693,E2 3284.693} C_VEL
LIN {X 0,Y 551.937,Z 989.03,A -85,B 0,C 180,E1 3289.951,E2 3289.951} C_VEL
LIN {X 0,Y 551.952,Z 989.03,A -85,B 0,C 180,E1 3295.1,E2 3295.1} C_VEL
LIN {X 0,Y 552.142,Z 989.428,A -85,B 0,C 180,E1 3300.628,E2 3300.628} C_VEL
LIN {X 0,Y 557.634,Z 1010.613,A -85,B 0,C 180,E1 3302.176,E2 3302.176} C_VEL
LIN {X 0,Y 556.306,Z 1044.957,A -85,B 0,C 180,E1 3304.644,E2 3304.644} C_VEL
LIN {X 0,Y 554.939,Z 1076.369,A -85,B 0,C 180,E1 3307.624,E2 3307.624} C_VEL
LIN {X 0,Y 553.871,Z 1103.029,A -85,B 0,C 180,E1 3310.918,E2 3310.918} C_VEL
LIN {X 0,Y 553.075,Z 1125.047,A -85,B 0,C 180,E1 3314.47,E2 3314.47} C_VEL
LIN {X 0,Y 552.66,Z 1142.156,A -85,B 0,C 180,E1 3318.184,E2 3318.184} C_VEL
LIN {X 0,Y 552.591,Z 1153.829,A -85,B 0,C 180,E1 3321.758,E2 3321.758} C_VEL
LIN {X 0,Y 552.463,Z 1161.027,A -85,B 0,C 180,E1 3325.3,E2 3325.3} C_VEL
LIN {X 0,Y 552.459,Z 1164.117,A -85,B 0,C 180,E1 3328.435,E2 3328.435} C_VEL
LIN {X 0,Y 552.591,Z 1164.058,A -85,B 0,C 180,E1 3331.565,E2 3331.565} C_VEL
LIN {X 0,Y 552.509,Z 1159.678,A -85,B 0,C 180,E1 3335.486,E2 3335.486} C_VEL
LIN {X 0,Y 552.622,Z 1150.171,A -85,B 0,C 180,E1 3339.43,E2 3339.43} C_VEL
LIN {X 0,Y 552.913,Z 1135.085,A -85,B 0,C 180,E1 3343.414,E2 3343.414} C_VEL
LIN {X 0,Y 553.481,Z 1113.374,A -85,B 0,C 180,E1 3347.452,E2 3347.452} C_VEL
LIN {X 0,Y 554.468,Z 1088.232,A -85,B 0,C 180,E1 3350.929,E2 3350.929} C_VEL
LIN {X 0,Y 555.736,Z 1058.96,A -85,B 0,C 180,E1 3354.036,E2 3354.036} C_VEL
LIN {X 0,Y 557.159,Z 1026.804,A -85,B 0,C 180,E1 3356.654,E2 3356.654} C_VEL
LIN {X 0,Y 557.482,Z 1006.769,A -85,B 0,C 180,E1 3357.99,E2 3357.99} C_VEL
LIN {X 0,Y 552.046,Z 989.03,A -85,B 0,C 180,E1 3359.342,E2 3359.342} C_VEL
LIN {X 0,Y 551.96,Z 989.03,A -85,B 0,C 180,E1 3365.039,E2 3365.039} C_VEL
LIN {X 0,Y 551.872,Z 989.03,A -85,B 0,C 180,E1 3371.015,E2 3371.015} C_VEL
LIN {X 0,Y 551.967,Z 989.03,A -85,B 0,C 180,E1 3376.887,E2 3376.887} C_VEL
LIN {X 0,Y 551.977,Z 989.03,A -85,B 0,C 180,E1 3383.029,E2 3383.029} C_VEL
LIN {X 0,Y 551.928,Z 989.03,A -85,B 0,C 180,E1 3388.705,E2 3388.705} C_VEL
LIN {X 0,Y 552.113,Z 989.03,A -85,B 0,C 180,E1 3394.416,E2 3394.416} C_VEL
LIN {X 0,Y 552.262,Z 989.03,A -85,B 0,C 180,E1 3400.86,E2 3400.86} C_VEL
LIN {X 0,Y 551.938,Z 989.03,A -85,B 0,C 180,E1 3405.756,E2 3405.756} C_VEL
LIN {X 0,Y 552.178,Z 989.03,A -85,B 0,C 180,E1 3410.563,E2 3410.563} C_VEL
LIN {X 0,Y 552.329,Z 989.03,A -85,B 0,C 180,E1 3415.299,E2 3415.299} C_VEL
LIN {X 0,Y 552.361,Z 989.03,A -85,B 0,C 180,E1 3420,E2 3420} C_VEL
LIN {X 0,Y 552.36,Z 989.03,A -85,B 0,C 180,E1 3424.701,E2 3424.701} C_VEL
LIN {X 0,Y 552.166,Z 989.03,A -85,B 0,C 180,E1 3430.31,E2 3430.31} C_VEL
LIN {X 0,Y 552.095,Z 989.03,A -85,B 0,C 180,E1 3436.121,E2 3436.121} C_VEL
LIN {X 0,Y 552.1,Z 989.03,A -85,B 0,C 180,E1 3439.635,E2 3439.635} C_VEL
LIN {X 0,Y 548.075,Z 989.03,A -85,B 0,C 180,E1 3441.404,E2 3441.404} C_VEL
LIN {X 0,Y 544.095,Z 989.03,A -85,B 0,C 180,E1 3443.198,E2 3443.198} C_VEL
LIN {X 0,Y 544.106,Z 989.03,A -85,B 0,C 180,E1 3448.129,E2 3448.129} C_VEL
LIN {X 0,Y 544.192,Z 989.03,A -85,B 0,C 180,E1 3453.706,E2 3453.706} C_VEL
LIN {X 0,Y 544.029,Z 989.03,A -85,B 0,C 180,E1 3459.638,E2 3459.638} C_VEL
LIN {X 0,Y 543.942,Z 989.03,A -85,B 0,C 180,E1 3466.159,E2 3466.159} C_VEL
LIN {X 0,Y 544.158,Z 989.03,A -85,B 0,C 180,E1 3472.404,E2 3472.404} C_VEL
LIN {X 0,Y 544.368,Z 989.03,A -85,B 0,C 180,E1 3476.261,E2 3476.261} C_VEL
LIN {X 0,Y 554.211,Z 1011.297,A -85,B 0,C 180,E1 3477.282,E2 3477.282} C_VEL
LIN {X 0,Y 553.636,Z 1079.08,A -85,B 0,C 180,E1 3478.398,E2 3478.398} C_VEL
LIN {X 0,Y 552.51,Z 1118.402,A -85,B 0,C 180,E1 3479.675,E2 3479.675} C_VEL
LIN {X 0,Y 550.882,Z 1157.188,A -85,B 0,C 180,E1 3481.626,E2 3481.626} C_VEL
LIN {X 0,Y 549.113,Z 1193.405,A -85,B 0,C 180,E1 3484.199,E2 3484.199} C_VEL
LIN {X 0,Y 547.566,Z 1224.032,A -85,B 0,C 180,E1 3487.091,E2 3487.091} C_VEL
LIN {X 0,Y 546.237,Z 1251.323,A -85,B 0,C 180,E1 3490.441,E2 3490.441} C_VEL
LIN {X 0,Y 545.291,Z 1274.261,A -85,B 0,C 180,E1 3494.14,E2 3494.14} C_VEL
LIN {X 0,Y 544.832,Z 1291.979,A -85,B 0,C 180,E1 3498.01,E2 3498.01} C_VEL
LIN {X 0,Y 544.713,Z 1303.716,A -85,B 0,C 180,E1 3501.637,E2 3501.637} C_VEL
LIN {X 0,Y 544.552,Z 1312.017,A -85,B 0,C 180,E1 3505.992,E2 3505.992} C_VEL
LIN {X 0,Y 544.564,Z 1314.5,A -85,B 0,C 180,E1 3509.999,E2 3509.999} C_VEL
LIN {X 0,Y 544.575,Z 1311.982,A -85,B 0,C 180,E1 3514.042,E2 3514.042} C_VEL
LIN {X 0,Y 544.78,Z 1303.719,A -85,B 0,C 180,E1 3518.361,E2 3518.361} C_VEL
LIN {X 0,Y 545.012,Z 1290.447,A -85,B 0,C 180,E1 3522.39,E2 3522.39} C_VEL
LIN {X 0,Y 545.561,Z 1271.211,A -85,B 0,C 180,E1 3526.424,E2 3526.424} C_VEL
LIN {X 0,Y 546.484,Z 1246.45,A -85,B 0,C 180,E1 3530.227,E2 3530.227} C_VEL
LIN {X 0,Y 547.852,Z 1218.013,A -85,B 0,C 180,E1 3533.539,E2 3533.539} C_VEL
LIN {X 0,Y 549.523,Z 1185.305,A -85,B 0,C 180,E1 3536.444,E2 3536.444} C_VEL
LIN {X 0,Y 551.151,Z 1150.946,A -85,B 0,C 180,E1 3538.734,E2 3538.734} C_VEL
LIN {X 0,Y 552.569,Z 1114.555,A -85,B 0,C 180,E1 3540.479,E2 3540.479} C_VEL
LIN {X 0,Y 553.718,Z 1077.357,A -85,B 0,C 180,E1 3541.637,E2 3541.637} C_VEL
LIN {X 0,Y 553.652,Z 1010.583,A -85,B 0,C 180,E1 3542.765,E2 3542.765} C_VEL
LIN {X 0,Y 543.984,Z 989.03,A -85,B 0,C 180,E1 3543.796,E2 3543.796} C_VEL
LIN {X 0,Y 544.075,Z 989.03,A -85,B 0,C 180,E1 3549.636,E2 3549.636} C_VEL
LIN {X 0,Y 544.013,Z 989.03,A -85,B 0,C 180,E1 3556.153,E2 3556.153} C_VEL
LIN {X 0,Y 544.088,Z 989.03,A -85,B 0,C 180,E1 3562.401,E2 3562.401} C_VEL
LIN {X 0,Y 544.034,Z 989.03,A -85,B 0,C 180,E1 3568.198,E2 3568.198} C_VEL
LIN {X 0,Y 544.102,Z 989.03,A -85,B 0,C 180,E1 3573.658,E2 3573.658} C_VEL
LIN {X 0,Y 544.197,Z 989.03,A -85,B 0,C 180,E1 3578.871,E2 3578.871} C_VEL
LIN {X 0,Y 544.227,Z 989.03,A -85,B 0,C 180,E1 3583.903,E2 3583.903} C_VEL
LIN {X 0,Y 544.286,Z 989.03,A -85,B 0,C 180,E1 3590.425,E2 3590.425} C_VEL
LIN {X 0,Y 544.432,Z 989.03,A -85,B 0,C 180,E1 3595.23,E2 3595.23} C_VEL
LIN {X 0,Y 544.432,Z 989.03,A -85,B 0,C 180,E1 3600,E2 3600} C_VEL
LIN {X 0,Y 544.422,Z 989.03,A -85,B 0,C 180,E1 3604.77,E2 3604.77} C_VEL
LIN {X 0,Y 544.38,Z 989.03,A -85,B 0,C 180,E1 3609.573,E2 3609.573} C_VEL
LIN {X 0,Y 544.307,Z 989.03,A -85,B 0,C 180,E1 3614.448,E2 3614.448} C_VEL
LIN {X 0,Y 544.228,Z 989.03,A -85,B 0,C 180,E1 3619.485,E2 3619.485} C_VEL
LIN {X 0,Y 544.095,Z 989.03,A -85,B 0,C 180,E1 3624.582,E2 3624.582} C_VEL
LIN {X 0,Y 544.003,Z 989.03,A -85,B 0,C 180,E1 3630.695,E2 3630.695} C_VEL
LIN {X 0,Y 543.933,Z 989.03,A -85,B 0,C 180,E1 3635.631,E2 3635.631} C_VEL
LIN {X 0,Y 543.935,Z 989.03,A -85,B 0,C 180,E1 3641.743,E2 3641.743} C_VEL
LIN {X 0,Y 544.05,Z 989.03,A -85,B 0,C 180,E1 3648.266,E2 3648.266} C_VEL
LIN {X 0,Y 543.998,Z 989.03,A -85,B 0,C 180,E1 3654.372,E2 3654.372} C_VEL
LIN {X 0,Y 544.222,Z 989.838,A -85,B 0,C 180,E1 3660.18,E2 3660.18} C_VEL
LIN {X 0,Y 550.413,Z 1012.629,A -85,B 0,C 180,E1 3661.912,E2 3661.912} C_VEL
LIN {X 0,Y 548.871,Z 1047.23,A -85,B 0,C 180,E1 3664.474,E2 3664.474} C_VEL
LIN {X 0,Y 547.318,Z 1078.699,A -85,B 0,C 180,E1 3667.557,E2 3667.557} C_VEL
LIN {X 0,Y 546.072,Z 1105.935,A -85,B 0,C 180,E1 3671.053,E2 3671.053} C_VEL
LIN {X 0,Y 545.224,Z 1127.762,A -85,B 0,C 180,E1 3674.757,E2 3674.757} C_VEL
LIN {X 0,Y 544.819,Z 1145.206,A -85,B 0,C 180,E1 3678.821,E2 3678.821} C_VEL
LIN {X 0,Y 544.706,Z 1156.705,A -85,B 0,C 180,E1 3682.839,E2 3682.839} C_VEL
LIN {X 0,Y 544.577,Z 1162.957,A -85,B 0,C 180,E1 3686.824,E2 3686.824} C_VEL
LIN {X 0,Y 544.563,Z 1164.497,A -85,B 0,C 180,E1 3690.001,E2 3690.001} C_VEL
LIN {X 0,Y 544.6,Z 1161.892,A -85,B 0,C 180,E1 3694.08,E2 3694.08} C_VEL
LIN {X 0,Y 544.776,Z 1153.601,A -85,B 0,C 180,E1 3698.362,E2 3698.362} C_VEL
LIN {X 0,Y 545.005,Z 1140.273,A -85,B 0,C 180,E1 3702.392,E2 3702.392} C_VEL
LIN {X 0,Y 545.55,Z 1120.95,A -85,B 0,C 180,E1 3706.425,E2 3706.425} C_VEL
LIN {X 0,Y 546.527,Z 1095.869,A -85,B 0,C 180,E1 3710.257,E2 3710.257} C_VEL
LIN {X 0,Y 547.931,Z 1066.522,A -85,B 0,C 180,E1 3713.645,E2 3713.645} C_VEL
LIN {X 0,Y 549.548,Z 1034.686,A -85,B 0,C 180,E1 3716.448,E2 3716.448} C_VEL
LIN {X 0,Y 549.951,Z 1008.198,A -85,B 0,C 180,E1 3718.315,E2 3718.315} C_VEL
LIN {X 0,Y 544.101,Z 989.03,A -85,B 0,C 180,E1 3719.828,E2 3719.828} C_VEL
LIN {X 0,Y 543.95,Z 989.03,A -85,B 0,C 180,E1 3725.633,E2 3725.633} C_VEL
LIN {X 0,Y 543.936,Z 989.03,A -85,B 0,C 180,E1 3731.746,E2 3731.746} C_VEL
LIN {X 0,Y 544.056,Z 989.03,A -85,B 0,C 180,E1 3738.268,E2 3738.268} C_VEL
LIN {X 0,Y 544.002,Z 989.03,A -85,B 0,C 180,E1 3744.374,E2 3744.374} C_VEL
LIN {X 0,Y 544.001,Z 989.03,A -85,B 0,C 180,E1 3750.048,E2 3750.048} C_VEL
LIN {X 0,Y 544.121,Z 989.03,A -85,B 0,C 180,E1 3755.419,E2 3755.419} C_VEL
LIN {X 0,Y 544.313,Z 989.03,A -85,B 0,C 180,E1 3760.57,E2 3760.57} C_VEL
LIN {X 0,Y 544.024,Z 989.03,A -85,B 0,C 180,E1 3766.129,E2 3766.129} C_VEL
LIN {X 0,Y 544.293,Z 989.03,A -85,B 0,C 180,E1 3770.425,E2 3770.425} C_VEL
LIN {X 0,Y 544.442,Z 989.03,A -85,B 0,C 180,E1 3775.231,E2 3775.231} C_VEL
LIN {X 0,Y 544.46,Z 989.03,A -85,B 0,C 180,E1 3780,E2 3780} C_VEL
LIN {X 0,Y 544.454,Z 989.03,A -85,B 0,C 180,E1 3784.769,E2 3784.769} C_VEL
LIN {X 0,Y 544.367,Z 989.03,A -85,B 0,C 180,E1 3789.574,E2 3789.574} C_VEL
LIN {X 0,Y 544.348,Z 989.03,A -85,B 0,C 180,E1 3794.447,E2 3794.447} C_VEL
LIN {X 0,Y 544.199,Z 989.03,A -85,B 0,C 180,E1 3799.623,E2 3799.623} C_VEL
LIN {X 0,Y 544.095,Z 989.03,A -85,B 0,C 180,E1 3803.198,E2 3803.198} C_VEL
LIN {X 0,Y 540.153,Z 989.03,A -85,B 0,C 180,E1 3805,E2 3805} C_VEL
LIN {X 0,Y 536.124,Z 989.03,A -85,B 0,C 180,E1 3806.829,E2 3806.829} C_VEL
LIN {X 0,Y 536.223,Z 989.03,A -85,B 0,C 180,E1 3812.408,E2 3812.408} C_VEL
LIN {X 0,Y 536.161,Z 989.03,A -85,B 0,C 180,E1 3818.255,E2 3818.255} C_VEL
LIN {X 0,Y 535.945,Z 989.03,A -85,B 0,C 180,E1 3824.738,E2 3824.738} C_VEL
LIN {X 0,Y 536.097,Z 989.03,A -85,B 0,C 180,E1 3829.653,E2 3829.653} C_VEL
LIN {X 0,Y 536.358,Z 989.216,A -85,B 0,C 180,E1 3835.699,E2 3835.699} C_VEL
LIN {X 0,Y 547.566,Z 1015.68,A -85,B 0,C 180,E1 3836.902,E2 3836.902} C_VEL
LIN {X 0,Y 546.878,Z 1080.953,A -85,B 0,C 180,E1 3838.008,E2 3838.008} C_VEL
LIN {X 0,Y 545.574,Z 1119.953,A -85,B 0,C 180,E1 3839.315,E2 3839.315} C_VEL
LIN {X 0,Y 543.804,Z 1156.982,A -85,B 0,C 180,E1 3841.209,E2 3841.209} C_VEL
LIN {X 0,Y 541.836,Z 1192.647,A -85,B 0,C 180,E1 3843.76,E2 3843.76} C_VEL
LIN {X 0,Y 540.093,Z 1224.031,A -85,B 0,C 180,E1 3846.755,E2 3846.755} C_VEL
LIN {X 0,Y 538.595,Z 1251.324,A -85,B 0,C 180,E1 3850.152,E2 3850.152} C_VEL
LIN {X 0,Y 537.476,Z 1274.262,A -85,B 0,C 180,E1 3853.903,E2 3853.903} C_VEL
LIN {X 0,Y 537.048,Z 1290.442,A -85,B 0,C 180,E1 3857.422,E2 3857.422} C_VEL
LIN {X 0,Y 536.815,Z 1303.716,A -85,B 0,C 180,E1 3861.513,E2 3861.513} C_VEL
LIN {X 0,Y 536.642,Z 1310.956,A -85,B 0,C 180,E1 3865.16,E2 3865.16} C_VEL
LIN {X 0,Y 536.668,Z 1314.087,A -85,B 0,C 180,E1 3868.388,E2 3868.388} C_VEL
LIN {X 0,Y 536.797,Z 1314.088,A -85,B 0,C 180,E1 3871.61,E2 3871.61} C_VEL
LIN {X 0,Y 536.755,Z 1309.756,A -85,B 0,C 180,E1 3875.646,E2 3875.646} C_VEL
LIN {X 0,Y 536.829,Z 1300.305,A -85,B 0,C 180,E1 3879.709,E2 3879.709} C_VEL
LIN {X 0,Y 537.255,Z 1284.761,A -85,B 0,C 180,E1 3883.937,E2 3883.937} C_VEL
LIN {X 0,Y 538.049,Z 1263.668,A -85,B 0,C 180,E1 3887.969,E2 3887.969} C_VEL
LIN {X 0,Y 539.338,Z 1237.543,A -85,B 0,C 180,E1 3891.676,E2 3891.676} C_VEL
LIN {X 0,Y 541.002,Z 1207.307,A -85,B 0,C 180,E1 3894.941,E2 3894.941} C_VEL
LIN {X 0,Y 542.883,Z 1173.532,A -85,B 0,C 180,E1 3897.701,E2 3897.701} C_VEL
LIN {X 0,Y 544.716,Z 1138.345,A -85,B 0,C 180,E1 3899.824,E2 3899.824} C_VEL
LIN {X 0,Y 546.199,Z 1101.757,A -85,B 0,C 180,E1 3901.373,E2 3901.373} C_VEL
LIN {X 0,Y 547.384,Z 1065.162,A -85,B 0,C 180,E1 3902.324,E2 3902.324} C_VEL
LIN {X 0,Y 547.014,Z 1013.199,A -85,B 0,C 180,E1 3903.174,E2 3903.174} C_VEL
LIN {X 0,Y 536.113,Z 989.03,A -85,B 0,C 180,E1 3904.386,E2 3904.386} C_VEL
LIN {X 0,Y 536.199,Z 989.03,A -85,B 0,C 180,E1 3908.253,E2 3908.253} C_VEL
LIN {X 0,Y 535.981,Z 989.03,A -85,B 0,C 180,E1 3914.736,E2 3914.736} C_VEL
LIN {X 0,Y 536.069,Z 989.03,A -85,B 0,C 180,E1 3919.653,E2 3919.653} C_VEL
LIN {X 0,Y 536.048,Z 989.03,A -85,B 0,C 180,E1 3924.722,E2 3924.722} C_VEL
LIN {X 0,Y 536.058,Z 989.03,A -85,B 0,C 180,E1 3930.768,E2 3930.768} C_VEL
LIN {X 0,Y 536.193,Z 989.03,A -85,B 0,C 180,E1 3936.797,E2 3936.797} C_VEL
LIN {X 0,Y 536.386,Z 989.03,A -85,B 0,C 180,E1 3941.974,E2 3941.974} C_VEL
LIN {X 0,Y 536.334,Z 989.03,A -85,B 0,C 180,E1 3948.642,E2 3948.642} C_VEL
LIN {X 0,Y 536.528,Z 989.03,A -85,B 0,C 180,E1 3955.16,E2 3955.16} C_VEL
LIN {X 0,Y 536.539,Z 989.03,A -85,B 0,C 180,E1 3960,E2 3960} C_VEL
LIN {X 0,Y 536.509,Z 989.03,A -85,B 0,C 180,E1 3964.84,E2 3964.84} C_VEL
LIN {X 0,Y 536.399,Z 989.03,A -85,B 0,C 180,E1 3970.062,E2 3970.062} C_VEL
LIN {X 0,Y 536.37,Z 989.03,A -85,B 0,C 180,E1 3974.666,E2 3974.666} C_VEL
LIN {X 0,Y 536.318,Z 989.03,A -85,B 0,C 180,E1 3979.732,E2 3979.732} C_VEL
LIN {X 0,Y 536.094,Z 989.03,A -85,B 0,C 180,E1 3985.745,E2 3985.745} C_VEL
LIN {X 0,Y 536.096,Z 989.03,A -85,B 0,C 180,E1 3990.441,E2 3990.441} C_VEL
LIN {X 0,Y 536.002,Z 989.03,A -85,B 0,C 180,E1 3996.241,E2 3996.241} C_VEL
LIN {X 0,Y 535.952,Z 989.03,A -85,B 0,C 180,E1 4002.509,E2 4002.509} C_VEL
LIN {X 0,Y 536.051,Z 989.03,A -85,B 0,C 180,E1 4007.499,E2 4007.499} C_VEL
LIN {X 0,Y 536.108,Z 989.03,A -85,B 0,C 180,E1 4013.766,E2 4013.766} C_VEL
LIN {X 0,Y 536.225,Z 989.283,A -85,B 0,C 180,E1 4019.66,E2 4019.66} C_VEL
LIN {X 0,Y 543.229,Z 1014.279,A -85,B 0,C 180,E1 4021.618,E2 4021.618} C_VEL
LIN {X 0,Y 541.443,Z 1049.456,A -85,B 0,C 180,E1 4024.296,E2 4024.296} C_VEL
LIN {X 0,Y 539.719,Z 1080.827,A -85,B 0,C 180,E1 4027.467,E2 4027.467} C_VEL
LIN {X 0,Y 538.326,Z 1108.644,A -85,B 0,C 180,E1 4031.195,E2 4031.195} C_VEL
LIN {X 0,Y 537.382,Z 1129.755,A -85,B 0,C 180,E1 4034.946,E2 4034.946} C_VEL
LIN {X 0,Y 536.947,Z 1145.204,A -85,B 0,C 180,E1 4038.655,E2 4038.655} C_VEL
LIN {X 0,Y 536.813,Z 1156.703,A -85,B 0,C 180,E1 4042.733,E2 4042.733} C_VEL
LIN {X 0,Y 536.683,Z 1162.957,A -85,B 0,C 180,E1 4046.777,E2 4046.777} C_VEL
LIN {X 0,Y 536.689,Z 1164.497,A -85,B 0,C 180,E1 4050.001,E2 4050.001} C_VEL
LIN {X 0,Y 536.681,Z 1162.862,A -85,B 0,C 180,E1 4053.224,E2 4053.224} C_VEL
LIN {X 0,Y 536.713,Z 1156.489,A -85,B 0,C 180,E1 4057.269,E2 4057.269} C_VEL
LIN {X 0,Y 536.944,Z 1144.876,A -85,B 0,C 180,E1 4061.346,E2 4061.346} C_VEL
LIN {X 0,Y 537.524,Z 1127.283,A -85,B 0,C 180,E1 4065.468,E2 4065.468} C_VEL
LIN {X 0,Y 538.459,Z 1103.851,A -85,B 0,C 180,E1 4069.439,E2 4069.439} C_VEL
LIN {X 0,Y 539.91,Z 1076.955,A -85,B 0,C 180,E1 4072.875,E2 4072.875} C_VEL
LIN {X 0,Y 541.659,Z 1045.919,A -85,B 0,C 180,E1 4075.916,E2 4075.916} C_VEL
LIN {X 0,Y 543.054,Z 1011.729,A -85,B 0,C 180,E1 4078.472,E2 4078.472} C_VEL
LIN {X 0,Y 536.157,Z 989.03,A -85,B 0,C 180,E1 4080.287,E2 4080.287} C_VEL
LIN {X 0,Y 536.022,Z 989.03,A -85,B 0,C 180,E1 4086.242,E2 4086.242} C_VEL
LIN {X 0,Y 535.952,Z 989.03,A -85,B 0,C 180,E1 4092.512,E2 4092.512} C_VEL
LIN {X 0,Y 536.056,Z 989.03,A -85,B 0,C 180,E1 4097.501,E2 4097.501} C_VEL
LIN {X 0,Y 536.113,Z 989.03,A -85,B 0,C 180,E1 4103.767,E2 4103.767} C_VEL
LIN {X 0,Y 536.094,Z 989.03,A -85,B 0,C 180,E1 4109.559,E2 4109.559} C_VEL
LIN {X 0,Y 536.173,Z 989.03,A -85,B 0,C 180,E1 4115.03,E2 4115.03} C_VEL
LIN {X 0,Y 536.388,Z 989.03,A -85,B 0,C 180,E1 4120.271,E2 4120.271} C_VEL
LIN {X 0,Y 536.162,Z 989.03,A -85,B 0,C 180,E1 4125.328,E2 4125.328} C_VEL
LIN {X 0,Y 536.373,Z 989.03,A -85,B 0,C 180,E1 4130.282,E2 4130.282} C_VEL
LIN {X 0,Y 536.539,Z 989.03,A -85,B 0,C 180,E1 4135.16,E2 4135.16} C_VEL
LIN {X 0,Y 536.59,Z 989.03,A -85,B 0,C 180,E1 4140,E2 4140} C_VEL
LIN {X 0,Y 536.54,Z 989.03,A -85,B 0,C 180,E1 4144.84,E2 4144.84} C_VEL
LIN {X 0,Y 536.419,Z 989.03,A -85,B 0,C 180,E1 4150.068,E2 4150.068} C_VEL
LIN {X 0,Y 536.403,Z 989.03,A -85,B 0,C 180,E1 4154.666,E2 4154.666} C_VEL
LIN {X 0,Y 536.309,Z 989.03,A -85,B 0,C 180,E1 4159.732,E2 4159.732} C_VEL
LIN {X 0,Y 536.094,Z 989.03,A -85,B 0,C 180,E1 4165.742,E2 4165.742} C_VEL
LIN {X 0,Y 536.124,Z 989.03,A -85,B 0,C 180,E1 4166.829,E2 4166.829} C_VEL
LIN {X 0,Y 532.063,Z 989.03,A -85,B 0,C 180,E1 4168.659,E2 4168.659} C_VEL
LIN {X 0,Y 528.168,Z 989.03,A -85,B 0,C 180,E1 4170.517,E2 4170.517} C_VEL
LIN {X 0,Y 528.315,Z 989.03,A -85,B 0,C 180,E1 4174.836,E2 4174.836} C_VEL
LIN {X 0,Y 528.084,Z 989.03,A -85,B 0,C 180,E1 4181.087,E2 4181.087} C_VEL
LIN {X 0,Y 528.046,Z 989.03,A -85,B 0,C 180,E1 4186.696,E2 4186.696} C_VEL
LIN {X 0,Y 528.29,Z 989.03,A -85,B 0,C 180,E1 4193.14,E2 4193.14} C_VEL
LIN {X 0,Y 528.392,Z 989.215,A -85,B 0,C 180,E1 4195.107,E2 4195.107} C_VEL
LIN {X 0,Y 540.944,Z 1018.076,A -85,B 0,C 180,E1 4196.481,E2 4196.481} C_VEL
LIN {X 0,Y 540.167,Z 1080.965,A -85,B 0,C 180,E1 4197.562,E2 4197.562} C_VEL
LIN {X 0,Y 538.689,Z 1120.673,A -85,B 0,C 180,E1 4198.914,E2 4198.914} C_VEL
LIN {X 0,Y 536.64,Z 1158.724,A -85,B 0,C 180,E1 4200.906,E2 4200.906} C_VEL
LIN {X 0,Y 534.505,Z 1193.908,A -85,B 0,C 180,E1 4203.486,E2 4203.486} C_VEL
LIN {X 0,Y 532.619,Z 1224.031,A -85,B 0,C 180,E1 4206.409,E2 4206.409} C_VEL
LIN {X 0,Y 530.963,Z 1251.104,A -85,B 0,C 180,E1 4209.822,E2 4209.822} C_VEL
LIN {X 0,Y 529.755,Z 1274.263,A -85,B 0,C 180,E1 4213.662,E2 4213.662} C_VEL
LIN {X 0,Y 529.14,Z 1291.98,A -85,B 0,C 180,E1 4217.649,E2 4217.649} C_VEL
LIN {X 0,Y 528.922,Z 1303.716,A -85,B 0,C 180,E1 4221.385,E2 4221.385} C_VEL
LIN {X 0,Y 528.754,Z 1310.956,A -85,B 0,C 180,E1 4225.088,E2 4225.088} C_VEL
LIN {X 0,Y 528.767,Z 1314.087,A -85,B 0,C 180,E1 4228.364,E2 4228.364} C_VEL
LIN {X 0,Y 528.741,Z 1313.393,A -85,B 0,C 180,E1 4232.753,E2 4232.753} C_VEL
LIN {X 0,Y 528.855,Z 1308.224,A -85,B 0,C 180,E1 4236.553,E2 4236.553} C_VEL
LIN {X 0,Y 528.955,Z 1298.373,A -85,B 0,C 180,E1 4240.488,E2 4240.488} C_VEL
LIN {X 0,Y 529.504,Z 1283.144,A -85,B 0,C 180,E1 4244.504,E2 4244.504} C_VEL
LIN {X 0,Y 530.406,Z 1262.345,A -85,B 0,C 180,E1 4248.451,E2 4248.451} C_VEL
LIN {X 0,Y 531.825,Z 1236.631,A -85,B 0,C 180,E1 4252.113,E2 4252.113} C_VEL
LIN {X 0,Y 533.593,Z 1207.615,A -85,B 0,C 180,E1 4255.281,E2 4255.281} C_VEL
LIN {X 0,Y 535.69,Z 1174.31,A -85,B 0,C 180,E1 4258.047,E2 4258.047} C_VEL
LIN {X 0,Y 537.766,Z 1138.151,A -85,B 0,C 180,E1 4260.26,E2 4260.26} C_VEL
LIN {X 0,Y 539.405,Z 1101.658,A -85,B 0,C 180,E1 4261.818,E2 4261.818} C_VEL
LIN {X 0,Y 540.702,Z 1063.959,A -85,B 0,C 180,E1 4262.795,E2 4262.795} C_VEL
LIN {X 0,Y 540.354,Z 1015.7,A -85,B 0,C 180,E1 4263.598,E2 4263.598} C_VEL
LIN {X 0,Y 528.213,Z 989.03,A -85,B 0,C 180,E1 4264.968,E2 4264.968} C_VEL
LIN {X 0,Y 528.099,Z 989.03,A -85,B 0,C 180,E1 4271.087,E2 4271.087} C_VEL
LIN {X 0,Y 528.092,Z 989.03,A -85,B 0,C 180,E1 4276.704,E2 4276.704} C_VEL
LIN {X 0,Y 528.192,Z 989.03,A -85,B 0,C 180,E1 4283.135,E2 4283.135} C_VEL
LIN {X 0,Y 528.156,Z 989.03,A -85,B 0,C 180,E1 4289.052,E2 4289.052} C_VEL
LIN {X 0,Y 528.261,Z 989.03,A -85,B 0,C 180,E1 4294.63,E2 4294.63} C_VEL
LIN {X 0,Y 528.443,Z 989.03,A -85,B 0,C 180,E1 4300.447,E2 4300.447} C_VEL
LIN {X 0,Y 528.202,Z 989.03,A -85,B 0,C 180,E1 4306.247,E2 4306.247} C_VEL
LIN {X 0,Y 528.443,Z 989.03,A -85,B 0,C 180,E1 4311.792,E2 4311.792} C_VEL
LIN {X 0,Y 528.647,Z 989.03,A -85,B 0,C 180,E1 4317.512,E2 4317.512} C_VEL
LIN {X 0,Y 528.736,Z 989.03,A -85,B 0,C 180,E1 4323.272,E2 4323.272} C_VEL
LIN {X 0,Y 528.535,Z 989.03,A -85,B 0,C 180,E1 4329.863,E2 4329.863} C_VEL
LIN {X 0,Y 528.46,Z 989.03,A -85,B 0,C 180,E1 4334.891,E2 4334.891} C_VEL
LIN {X 0,Y 528.384,Z 989.03,A -85,B 0,C 180,E1 4340.041,E2 4340.041} C_VEL
LIN {X 0,Y 528.217,Z 989.03,A -85,B 0,C 180,E1 4345.372,E2 4345.372} C_VEL
LIN {X 0,Y 528.14,Z 989.03,A -85,B 0,C 180,E1 4351.001,E2 4351.001} C_VEL
LIN {X 0,Y 528.054,Z 989.03,A -85,B 0,C 180,E1 4356.876,E2 4356.876} C_VEL
LIN {X 0,Y 528.012,Z 989.03,A -85,B 0,C 180,E1 4363.304,E2 4363.304} C_VEL
LIN {X 0,Y 528.12,Z 989.03,A -85,B 0,C 180,E1 4368.915,E2 4368.915} C_VEL
LIN {X 0,Y 528.126,Z 989.03,A -85,B 0,C 180,E1 4375.149,E2 4375.149} C_VEL
LIN {X 0,Y 528.278,Z 989.189,A -85,B 0,C 180,E1 4379.15,E2 4379.15} C_VEL
LIN {X 0,Y 535.989,Z 1017.296,A -85,B 0,C 180,E1 4381.406,E2 4381.406} C_VEL
LIN {X 0,Y 533.953,Z 1052.802,A -85,B 0,C 180,E1 4384.223,E2 4384.223} C_VEL
LIN {X 0,Y 532.03,Z 1083.302,A -85,B 0,C 180,E1 4387.434,E2 4387.434} C_VEL
LIN {X 0,Y 530.579,Z 1109.975,A -85,B 0,C 180,E1 4391.125,E2 4391.125} C_VEL
LIN {X 0,Y 529.561,Z 1131.709,A -85,B 0,C 180,E1 4395.141,E2 4395.141} C_VEL
LIN {X 0,Y 529.12,Z 1148.164,A -85,B 0,C 180,E1 4399.405,E2 4399.405} C_VEL
LIN {X 0,Y 528.906,Z 1158.309,A -85,B 0,C 180,E1 4403.448,E2 4403.448} C_VEL
LIN {X 0,Y 528.765,Z 1163.388,A -85,B 0,C 180,E1 4407.193,E2 4407.193} C_VEL
LIN {X 0,Y 528.904,Z 1164.06,A -85,B 0,C 180,E1 4411.636,E2 4411.636} C_VEL
LIN {X 0,Y 528.829,Z 1159.682,A -85,B 0,C 180,E1 4415.732,E2 4415.732} C_VEL
LIN {X 0,Y 528.973,Z 1150.178,A -85,B 0,C 180,E1 4419.856,E2 4419.856} C_VEL
LIN {X 0,Y 529.418,Z 1134.549,A -85,B 0,C 180,E1 4424.153,E2 4424.153} C_VEL
LIN {X 0,Y 530.371,Z 1113.383,A -85,B 0,C 180,E1 4428.239,E2 4428.239} C_VEL
LIN {X 0,Y 531.781,Z 1087.49,A -85,B 0,C 180,E1 4431.962,E2 4431.962} C_VEL
LIN {X 0,Y 533.6,Z 1058.093,A -85,B 0,C 180,E1 4435.188,E2 4435.188} C_VEL
LIN {X 0,Y 535.645,Z 1025.528,A -85,B 0,C 180,E1 4437.914,E2 4437.914} C_VEL
LIN {X 0,Y 535.591,Z 1013.181,A -85,B 0,C 180,E1 4438.808,E2 4438.808} C_VEL
LIN {X 0,Y 528.226,Z 989.03,A -85,B 0,C 180,E1 4440.823,E2 4440.823} C_VEL
LIN {X 0,Y 528.078,Z 989.03,A -85,B 0,C 180,E1 4446.877,E2 4446.877} C_VEL
LIN {X 0,Y 528.012,Z 989.03,A -85,B 0,C 180,E1 4453.307,E2 4453.307} C_VEL
LIN {X 0,Y 528.127,Z 989.03,A -85,B 0,C 180,E1 4458.917,E2 4458.917} C_VEL
LIN {X 0,Y 528.123,Z 989.03,A -85,B 0,C 180,E1 4465.15,E2 4465.15} C_VEL
LIN {X 0,Y 528.185,Z 989.03,A -85,B 0,C 180,E1 4470.944,E2 4470.944} C_VEL
LIN {X 0,Y 528.257,Z 989.03,A -85,B 0,C 180,E1 4476.428,E2 4476.428} C_VEL
LIN {X 0,Y 528.475,Z 989.03,A -85,B 0,C 180,E1 4481.695,E2 4481.695} C_VEL
LIN {X 0,Y 528.396,Z 989.03,A -85,B 0,C 180,E1 4488.469,E2 4488.469} C_VEL
LIN {X 0,Y 528.689,Z 989.03,A -85,B 0,C 180,E1 4493.445,E2 4493.445} C_VEL
LIN {X 0,Y 528.689,Z 989.03,A -85,B 0,C 180,E1 4500,E2 4500} C_VEL
LIN {X 0,Y 528.637,Z 989.03,A -85,B 0,C 180,E1 4504.912,E2 4504.912} C_VEL
LIN {X 0,Y 528.539,Z 989.03,A -85,B 0,C 180,E1 4509.863,E2 4509.863} C_VEL
LIN {X 0,Y 528.485,Z 989.03,A -85,B 0,C 180,E1 4514.89,E2 4514.89} C_VEL
LIN {X 0,Y 528.378,Z 989.03,A -85,B 0,C 180,E1 4520.041,E2 4520.041} C_VEL
LIN {X 0,Y 528.215,Z 989.03,A -85,B 0,C 180,E1 4525.373,E2 4525.373} C_VEL
LIN {X 0,Y 528.168,Z 989.03,A -85,B 0,C 180,E1 4530.517,E2 4530.517} C_VEL
LIN {X 0,Y 525.716,Z 989.03,A -85,B 0,C 180,E1 4531.92,E2 4531.92} C_VEL
LIN {X 0,Y 520.285,Z 989.03,A -85,B 0,C 180,E1 4534.266,E2 4534.266} C_VEL
LIN {X 0,Y 520.224,Z 989.03,A -85,B 0,C 180,E1 4539.652,E2 4539.652} C_VEL
LIN {X 0,Y 520.115,Z 989.03,A -85,B 0,C 180,E1 4545.867,E2 4545.867} C_VEL
LIN {X 0,Y 520.269,Z 989.03,A -85,B 0,C 180,E1 4551.544,E2 4551.544} C_VEL
LIN {X 0,Y 520.467,Z 989.238,A -85,B 0,C 180,E1 4554.5,E2 4554.5} C_VEL
LIN {X 0,Y 534.337,Z 1020.133,A -85,B 0,C 180,E1 4556.043,E2 4556.043} C_VEL
LIN {X 0,Y 533.498,Z 1080.965,A -85,B 0,C 180,E1 4557.106,E2 4557.106} C_VEL
LIN {X 0,Y 531.923,Z 1119.87,A -85,B 0,C 180,E1 4558.435,E2 4558.435} C_VEL
LIN {X 0,Y 529.707,Z 1157.59,A -85,B 0,C 180,E1 4560.41,E2 4560.41} C_VEL
LIN {X 0,Y 527.348,Z 1192.642,A -85,B 0,C 180,E1 4562.982,E2 4562.982} C_VEL
LIN {X 0,Y 525.143,Z 1224.149,A -85,B 0,C 180,E1 4566.067,E2 4566.067} C_VEL
LIN {X 0,Y 523.323,Z 1251.386,A -85,B 0,C 180,E1 4569.556,E2 4569.556} C_VEL
LIN {X 0,Y 521.986,Z 1274.265,A -85,B 0,C 180,E1 4573.412,E2 4573.412} C_VEL
LIN {X 0,Y 521.384,Z 1290.443,A -85,B 0,C 180,E1 4577.037,E2 4577.037} C_VEL
LIN {X 0,Y 521.053,Z 1303.716,A -85,B 0,C 180,E1 4581.254,E2 4581.254} C_VEL
LIN {X 0,Y 520.858,Z 1310.956,A -85,B 0,C 180,E1 4585.013,E2 4585.013} C_VEL
LIN {X 0,Y 520.881,Z 1314.087,A -85,B 0,C 180,E1 4588.339,E2 4588.339} C_VEL
LIN {X 0,Y 520.994,Z 1314.089,A -85,B 0,C 180,E1 4591.659,E2 4591.659} C_VEL
LIN {X 0,Y 520.992,Z 1309.756,A -85,B 0,C 180,E1 4595.818,E2 4595.818} C_VEL
LIN {X 0,Y 521.071,Z 1300.126,A -85,B 0,C 180,E1 4600.072,E2 4600.072} C_VEL
LIN {X 0,Y 521.598,Z 1285.257,A -85,B 0,C 180,E1 4604.243,E2 4604.243} C_VEL
LIN {X 0,Y 522.635,Z 1263.665,A -85,B 0,C 180,E1 4608.518,E2 4608.518} C_VEL
LIN {X 0,Y 524.241,Z 1237.272,A -85,B 0,C 180,E1 4612.368,E2 4612.368} C_VEL
LIN {X 0,Y 526.291,Z 1207.175,A -85,B 0,C 180,E1 4615.7,E2 4615.7} C_VEL
LIN {X 0,Y 528.612,Z 1173.731,A -85,B 0,C 180,E1 4618.5,E2 4618.5} C_VEL
LIN {X 0,Y 530.886,Z 1137.866,A -85,B 0,C 180,E1 4620.71,E2 4620.71} C_VEL
LIN {X 0,Y 532.678,Z 1101.363,A -85,B 0,C 180,E1 4622.278,E2 4622.278} C_VEL
LIN {X 0,Y 534.118,Z 1062.734,A -85,B 0,C 180,E1 4623.274,E2 4623.274} C_VEL
LIN {X 0,Y 533.963,Z 1018.807,A -85,B 0,C 180,E1 4624.005,E2 4624.005} C_VEL
LIN {X 0,Y 520.541,Z 990.825,A -85,B 0,C 180,E1 4625.469,E2 4625.469} C_VEL
LIN {X 0,Y 520.332,Z 989.03,A -85,B 0,C 180,E1 4625.578,E2 4625.578} C_VEL
LIN {X 0,Y 520.148,Z 989.03,A -85,B 0,C 180,E1 4631.855,E2 4631.855} C_VEL
LIN {X 0,Y 520.19,Z 989.03,A -85,B 0,C 180,E1 4638.151,E2 4638.151} C_VEL
LIN {X 0,Y 520.197,Z 989.03,A -85,B 0,C 180,E1 4644.314,E2 4644.314} C_VEL
LIN {X 0,Y 520.239,Z 989.03,A -85,B 0,C 180,E1 4650.479,E2 4650.479} C_VEL
LIN {X 0,Y 520.339,Z 989.03,A -85,B 0,C 180,E1 4656.047,E2 4656.047} C_VEL
LIN {X 0,Y 520.532,Z 989.03,A -85,B 0,C 180,E1 4661.405,E2 4661.405} C_VEL
LIN {X 0,Y 520.309,Z 989.03,A -85,B 0,C 180,E1 4666.585,E2 4666.585} C_VEL
LIN {X 0,Y 520.531,Z 989.03,A -85,B 0,C 180,E1 4671.666,E2 4671.666} C_VEL
LIN {X 0,Y 520.668,Z 989.03,A -85,B 0,C 180,E1 4676.677,E2 4676.677} C_VEL
LIN {X 0,Y 520.662,Z 989.03,A -85,B 0,C 180,E1 4681.661,E2 4681.661} C_VEL
LIN {X 0,Y 520.623,Z 989.03,A -85,B 0,C 180,E1 4686.657,E2 4686.657} C_VEL
LIN {X 0,Y 520.552,Z 989.03,A -85,B 0,C 180,E1 4691.707,E2 4691.707} C_VEL
LIN {X 0,Y 520.489,Z 989.03,A -85,B 0,C 180,E1 4696.916,E2 4696.916} C_VEL
LIN {X 0,Y 520.406,Z 989.03,A -85,B 0,C 180,E1 4702.144,E2 4702.144} C_VEL
LIN {X 0,Y 520.281,Z 989.03,A -85,B 0,C 180,E1 4707.648,E2 4707.648} C_VEL
LIN {X 0,Y 520.241,Z 989.03,A -85,B 0,C 180,E1 4713.442,E2 4713.442} C_VEL
LIN {X 0,Y 520.102,Z 989.03,A -85,B 0,C 180,E1 4719.663,E2 4719.663} C_VEL
LIN {X 0,Y 520.172,Z 989.03,A -85,B 0,C 180,E1 4725.875,E2 4725.875} C_VEL
LIN {X 0,Y 520.213,Z 989.03,A -85,B 0,C 180,E1 4731.552,E2 4731.552} C_VEL
LIN {X 0,Y 520.231,Z 989.03,A -85,B 0,C 180,E1 4737.262,E2 4737.262} C_VEL
LIN {X 0,Y 520.31,Z 989.6,A -85,B 0,C 180,E1 4738.649,E2 4738.649} C_VEL
LIN {X 0,Y 528.832,Z 1018.771,A -85,B 0,C 180,E1 4741.091,E2 4741.091} C_VEL
LIN {X 0,Y 526.536,Z 1054.184,A -85,B 0,C 180,E1 4743.97,E2 4743.97} C_VEL
LIN {X 0,Y 524.46,Z 1083.906,A -85,B 0,C 180,E1 4747.168,E2 4747.168} C_VEL
LIN {X 0,Y 522.825,Z 1109.969,A -85,B 0,C 180,E1 4750.834,E2 4750.834} C_VEL
LIN {X 0,Y 521.744,Z 1129.75,A -85,B 0,C 180,E1 4754.483,E2 4754.483} C_VEL
LIN {X 0,Y 521.217,Z 1146.544,A -85,B 0,C 180,E1 4758.732,E2 4758.732} C_VEL
LIN {X 0,Y 521.026,Z 1156.701,A -85,B 0,C 180,E1 4762.512,E2 4762.512} C_VEL
LIN {X 0,Y 520.879,Z 1162.956,A -85,B 0,C 180,E1 4766.679,E2 4766.679} C_VEL
LIN {X 0,Y 520.895,Z 1164.497,A -85,B 0,C 180,E1 4770.001,E2 4770.001} C_VEL
LIN {X 0,Y 520.883,Z 1162.864,A -85,B 0,C 180,E1 4773.322,E2 4773.322} C_VEL
LIN {X 0,Y 520.949,Z 1156.493,A -85,B 0,C 180,E1 4777.49,E2 4777.49} C_VEL
LIN {X 0,Y 521.245,Z 1144.88,A -85,B 0,C 180,E1 4781.693,E2 4781.693} C_VEL
LIN {X 0,Y 521.945,Z 1127.288,A -85,B 0,C 180,E1 4785.942,E2 4785.942} C_VEL
LIN {X 0,Y 523.058,Z 1105.311,A -85,B 0,C 180,E1 4789.816,E2 4789.816} C_VEL
LIN {X 0,Y 524.945,Z 1077.474,A -85,B 0,C 180,E1 4793.507,E2 4793.507} C_VEL
LIN {X 0,Y 527.068,Z 1045.931,A -85,B 0,C 180,E1 4796.689,E2 4796.689} C_VEL
LIN {X 0,Y 528.486,Z 1015.971,A -85,B 0,C 180,E1 4799.04,E2 4799.04} C_VEL
LIN {X 0,Y 520.287,Z 989.03,A -85,B 0,C 180,E1 4801.352,E2 4801.352} C_VEL
LIN {X 0,Y 520.082,Z 989.03,A -85,B 0,C 180,E1 4807.541,E2 4807.541} C_VEL
LIN {X 0,Y 520.108,Z 989.03,A -85,B 0,C 180,E1 4813.506,E2 4813.506} C_VEL
LIN {X 0,Y 520.223,Z 989.03,A -85,B 0,C 180,E1 4818.955,E2 4818.955} C_VEL
LIN {X 0,Y 520.178,Z 989.03,A -85,B 0,C 180,E1 4824.538,E2 4824.538} C_VEL
LIN {X 0,Y 520.255,Z 989.03,A -85,B 0,C 180,E1 4830.478,E2 4830.478} C_VEL
LIN {X 0,Y 520.347,Z 989.03,A -85,B 0,C 180,E1 4836.047,E2 4836.047} C_VEL
LIN {X 0,Y 520.562,Z 989.03,A -85,B 0,C 180,E1 4841.406,E2 4841.406} C_VEL
LIN {X 0,Y 520.473,Z 989.03,A -85,B 0,C 180,E1 4848.291,E2 4848.291} C_VEL
LIN {X 0,Y 520.762,Z 989.03,A -85,B 0,C 180,E1 4853.344,E2 4853.344} C_VEL
LIN {X 0,Y 520.937,Z 989.03,A -85,B 0,C 180,E1 4858.34,E2 4858.34} C_VEL
LIN {X 0,Y 520.723,Z 989.03,A -85,B 0,C 180,E1 4864.987,E2 4864.987} C_VEL
LIN {X 0,Y 520.635,Z 989.03,A -85,B 0,C 180,E1 4870.014,E2 4870.014} C_VEL
LIN {X 0,Y 520.546,Z 989.03,A -85,B 0,C 180,E1 4875.123,E2 4875.123} C_VEL
LIN {X 0,Y 520.434,Z 989.03,A -85,B 0,C 180,E1 4880.361,E2 4880.361} C_VEL
LIN {X 0,Y 520.257,Z 989.03,A -85,B 0,C 180,E1 4885.951,E2 4885.951} C_VEL
LIN {X 0,Y 520.308,Z 989.03,A -85,B 0,C 180,E1 4891.468,E2 4891.468} C_VEL
LIN {X 0,Y 520.285,Z 989.03,A -85,B 0,C 180,E1 4894.266,E2 4894.266} C_VEL
LIN {X 0,Y 518.993,Z 989.03,A -85,B 0,C 180,E1 4895.219,E2 4895.219} C_VEL
LIN {X 0,Y 512.416,Z 989.03,A -85,B 0,C 180,E1 4897.815,E2 4897.815} C_VEL
LIN {X 0,Y 512.33,Z 989.03,A -85,B 0,C 180,E1 4898.061,E2 4898.061} C_VEL
LIN {X 0,Y 512.191,Z 989.03,A -85,B 0,C 180,E1 4902.656,E2 4902.656} C_VEL
LIN {X 0,Y 512.317,Z 989.03,A -85,B 0,C 180,E1 4909.608,E2 4909.608} C_VEL
LIN {X 0,Y 512.511,Z 989.03,A -85,B 0,C 180,E1 4913.859,E2 4913.859} C_VEL
LIN {X 0,Y 527.771,Z 1022.193,A -85,B 0,C 180,E1 4915.595,E2 4915.595} C_VEL
LIN {X 0,Y 526.843,Z 1081.387,A -85,B 0,C 180,E1 4916.65,E2 4916.65} C_VEL
LIN {X 0,Y 525.138,Z 1119.869,A -85,B 0,C 180,E1 4917.979,E2 4917.979} C_VEL
LIN {X 0,Y 522.709,Z 1157.975,A -85,B 0,C 180,E1 4920.001,E2 4920.001} C_VEL
LIN {X 0,Y 520.131,Z 1192.639,A -85,B 0,C 180,E1 4922.576,E2 4922.576} C_VEL
LIN {X 0,Y 517.695,Z 1224.318,A -85,B 0,C 180,E1 4925.721,E2 4925.721} C_VEL
LIN {X 0,Y 515.73,Z 1251.244,A -85,B 0,C 180,E1 4929.22,E2 4929.22} C_VEL
